(* LS Electric XG5000 project: OnlineHelp_ECAT_Example *)
(* This project contains various examples from the online help topics. *)
(* PLC LSPLC *)
(* module base 0 slot 0: Input/Output Module:XEM-DN/DP32HP (DC 24V Input, Transistor Output, 32 Contacts) *)
(* module base 0 slot 1: Internal Positioning:XBF-PO06E (Open Collector Type, 6 Axis) *)
(* module base 0 slot 2: Positioning Module:XBF-PN08B (Position Control, EtherCAT Network Type(8 axis)) *)
VAR_GLOBAL
    _0002_A1_RDY AT %UX0.2.0 : BOOL; (* Positioning Module: 1-Axis Ready *)
    _0002_A2_RDY AT %UX0.2.1 : BOOL; (* Positioning Module: 2-Axis Ready *)
    _0002_A3_RDY AT %UX0.2.2 : BOOL; (* Positioning Module: 3-Axis Ready *)
    _0002_A4_RDY AT %UX0.2.3 : BOOL; (* Positioning Module: 4-Axis Ready *)
    _0002_LINKUP_INFO AT %UX0.2.14 : BOOL; (* Positioning Module: Link up/down information *)
END_VAR

PROGRAM LP606_XPM_ECON_DCON_Example (* task: Scan Program *)
VAR
    Connect_Servos : BOOL; (* command to connect to ECAT servos *)
    DCON_FB : XPM_DCON; (* EtherCAT disconnect function block *)
    Disconnect_Servos : BOOL; (* Disconnect from ECAT servos *)
    ECON_FB : XPM_ECON; (* EtherCAT Connect function block. *)
END_VAR

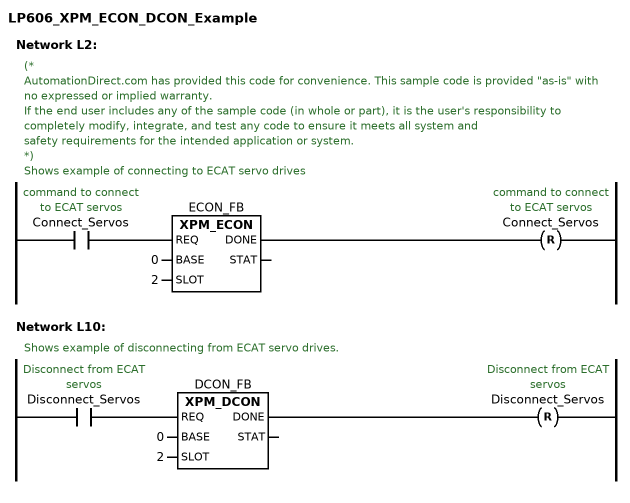
(* ( * / AutomationDirect.com has provided this code for convenience. This sample code is provided "as-is" with no expressed or implied warranty. / If the end user includes any of the sample code (in whole or part), it is the user's responsibility to completely modify, integrate, and test any code to ensure it meets all system and / safety requirements for the intended application or system. / * ) *)
(* Shows example of connecting to ECAT servo drives *)
(* Rung L2 *)
ECON_FB(REQ := Connect_Servos, BASE := 0, SLOT := 2);
IF ECON_FB.DONE THEN Connect_Servos := FALSE; END_IF;
(* Shows example of disconnecting from ECAT servo drives. *)
(* Rung L10 *)
DCON_FB(REQ := Disconnect_Servos, BASE := 0, SLOT := 2);
IF DCON_FB.DONE THEN Disconnect_Servos := FALSE; END_IF;
END_PROGRAM

PROGRAM LP607_XPM_SVON_SVOFF_Example (* task: Scan Program *)
(* This is an example for LP605 *)
VAR
    Axis1_SVOFF : XPM_SVOFF; (* function block for axis 1 servo off *)
    Axis1_SVOFF_Cmd : BOOL; (* axis 1 servo off command *)
    Axis1_SVON : XPM_SVON; (* SVON fb for axis 1 *)
    Axis1_SVON_Cmd : BOOL; (* axis 1 servo on command *)
END_VAR
VAR_EXTERNAL
    _0002_A1_RDY : BOOL; (* AT %UX0.2.0 *) (* Positioning Module: 1-Axis Ready *)
    _0002_LINKUP_INFO : BOOL; (* AT %UX0.2.14 *) (* Positioning Module: Link up/down information *)
END_VAR

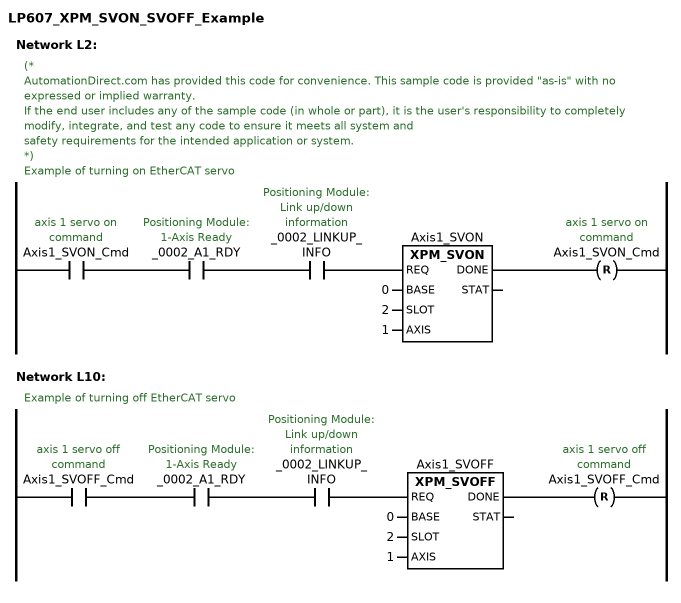
(* ( * / AutomationDirect.com has provided this code for convenience. This sample code is provided "as-is" with no expressed or implied warranty. / If the end user includes any of the sample code (in whole or part), it is the user's responsibility to completely modify, integrate, and test any code to ensure it meets all system and / safety requirements for the intended application or system. / * ) *)
(* Example of turning on EtherCAT servo *)
(* Rung L2 *)
Axis1_SVON(REQ := Axis1_SVON_Cmd AND _0002_A1_RDY AND _0002_LINKUP_INFO, BASE := 0, SLOT := 2, AXIS := 1);
IF Axis1_SVON.DONE THEN Axis1_SVON_Cmd := FALSE; END_IF;
(* Example of turning off EtherCAT servo *)
(* Rung L10 *)
Axis1_SVOFF(REQ := Axis1_SVOFF_Cmd AND _0002_A1_RDY AND _0002_LINKUP_INFO, BASE := 0, SLOT := 2, AXIS := 1);
IF Axis1_SVOFF.DONE THEN Axis1_SVOFF_Cmd := FALSE; END_IF;
END_PROGRAM

PROGRAM LP608_XPM_SVERD_SRST_Example (* task: Scan Program *)
(* this is an example of XPM_SVERD and XPM_SRST function blocks *)
VAR
    Axis1_Error : UINT; (* store axis 1 error *)
    Axis1_SRST : XPM_SRST; (* XPM_SRST for axis 1 *)
    Axis1_SVERD : XPM_SVERD; (* servo error reading for axis 1 *)
    Read_Axis1_Error : BOOL; (* command to read axis 1 error *)
    Reset_Axis1_Error : BOOL; (* reset command for axis error *)
END_VAR

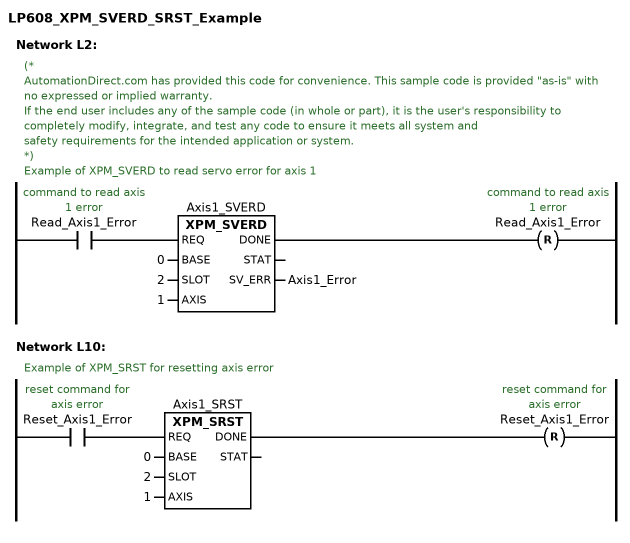
(* ( * / AutomationDirect.com has provided this code for convenience. This sample code is provided "as-is" with no expressed or implied warranty. / If the end user includes any of the sample code (in whole or part), it is the user's responsibility to completely modify, integrate, and test any code to ensure it meets all system and / safety requirements for the intended application or system. / * ) *)
(* Example of XPM_SVERD to read servo error for axis 1 *)
(* Rung L2 *)
Axis1_SVERD(REQ := Read_Axis1_Error, BASE := 0, SLOT := 2, AXIS := 1, SV_ERR => Axis1_Error);
IF Axis1_SVERD.DONE THEN Read_Axis1_Error := FALSE; END_IF;
(* Example of XPM_SRST for resetting axis error *)
(* Rung L10 *)
Axis1_SRST(REQ := Reset_Axis1_Error, BASE := 0, SLOT := 2, AXIS := 1);
IF Axis1_SRST.DONE THEN Reset_Axis1_Error := FALSE; END_IF;
END_PROGRAM

PROGRAM LP611_XPM_ENCRD_Example (* task: Scan Program *)
(* example for LP607 encoder reading *)
VAR
    Encoder_FB : XPM_ENCRD; (* reading encoder value *)
    Encoder_Value : DINT; (* encoder value from the read *)
    Read_Encoder_Value : BOOL; (* command to read encoder value. *)
END_VAR
VAR_EXTERNAL
    _0002_A1_RDY : BOOL; (* AT %UX0.2.0 *) (* Positioning Module: 1-Axis Ready *)
    _0002_LINKUP_INFO : BOOL; (* AT %UX0.2.14 *) (* Positioning Module: Link up/down information *)
END_VAR

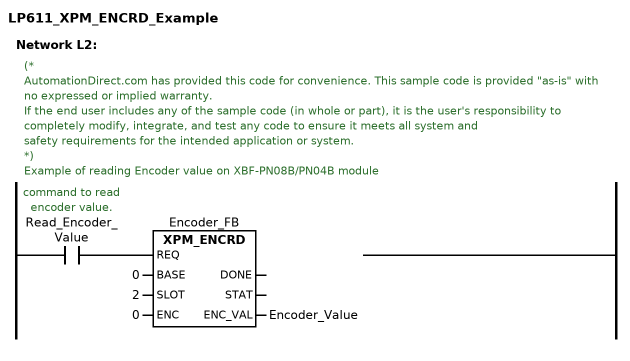
(* ( * / AutomationDirect.com has provided this code for convenience. This sample code is provided "as-is" with no expressed or implied warranty. / If the end user includes any of the sample code (in whole or part), it is the user's responsibility to completely modify, integrate, and test any code to ensure it meets all system and / safety requirements for the intended application or system. / * ) *)
(* Example of reading Encoder value on XBF-PN08B/PN04B module *)
(* Rung L2 *)
Encoder_FB(REQ := Read_Encoder_Value, BASE := 0, SLOT := 2, ENC := 0, ENC_VAL => Encoder_Value);
END_PROGRAM

PROGRAM LP612_XPM_TRQ_Example (* task: Scan Program *)
(* this is an example of XPM_TRQ *)
VAR
    Axes_SVOFF_Cmd : BOOL; (* axis 1 servo off command *)
    Axes_SVON_Cmd : BOOL; (* axes servo on command *)
    Axis1_Home : XPM_FLT; (* direct home of axis 1 *)
    Axis1_SVOFF : XPM_SVOFF; (* function block for axis 1 servo off *)
    Axis1_SVON : XPM_SVON; (* SVON fb for axis 1 *)
    Axis1_Torque_Time : UINT; (* gradient time for axis 1 torque fb *)
    Axis1_Torque_Value : INT; (* torque value for axis 1 *)
    Connect_Servos : BOOL; (* command to connect to ECAT servos *)
    DCON_FB : XPM_DCON; (* EtherCAT disconnect FB *)
    Disconnect_Servos : BOOL; (* Disconnect from ECAT servos *)
    ECON_FB : XPM_ECON; (* EtherCAT connect FB *)
    Execute_Torque_Control : BOOL; (* command to execute torque control *)
    Home_Axes : BOOL; (* home the axes *)
    TorqueCtrl_FB : XPM_TRQ; (* torque control fb for axis 1 *)
END_VAR
VAR_EXTERNAL
    _0002_A1_RDY : BOOL; (* AT %UX0.2.0 *) (* Positioning Module: 1-Axis Ready *)
    _0002_A4_RDY : BOOL; (* AT %UX0.2.3 *) (* Positioning Module: 4-Axis Ready *)
    _0002_LINKUP_INFO : BOOL; (* AT %UX0.2.14 *) (* Positioning Module: Link up/down information *)
END_VAR

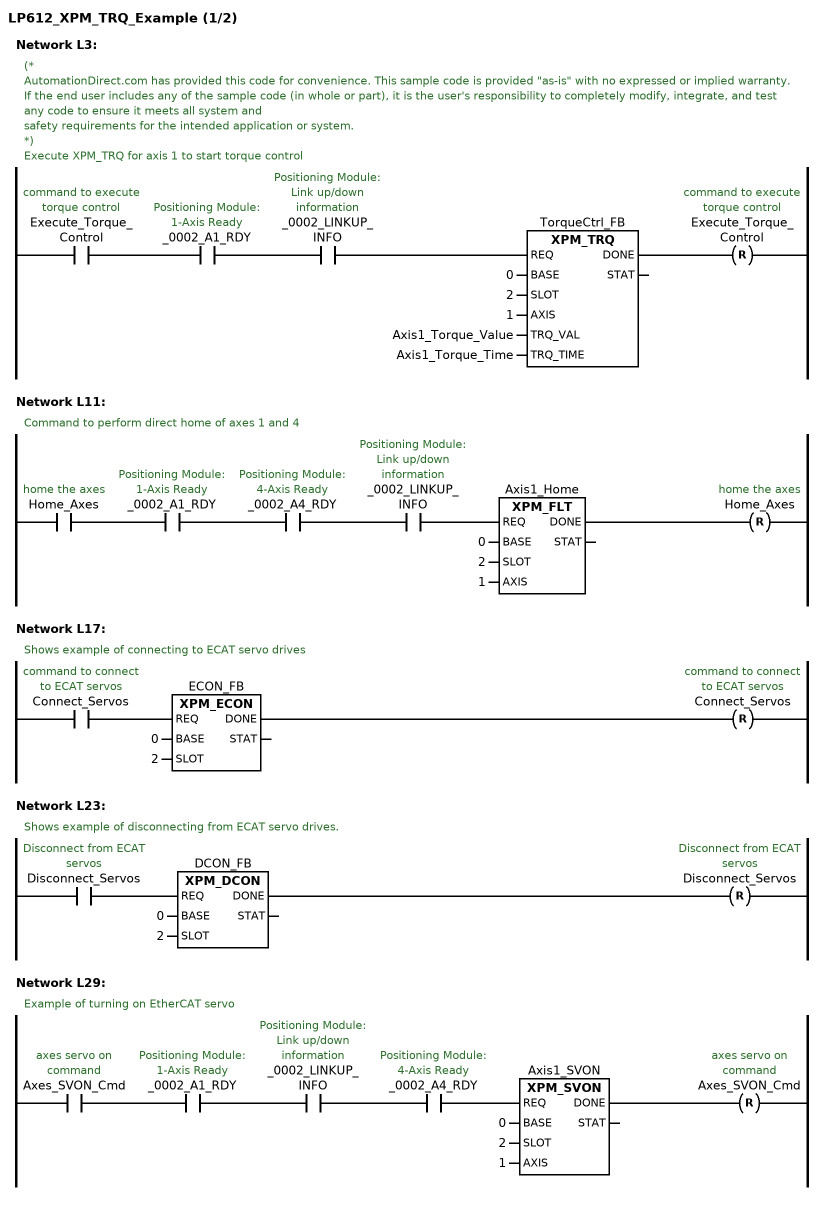
(* ( * / AutomationDirect.com has provided this code for convenience. This sample code is provided "as-is" with no expressed or implied warranty. / If the end user includes any of the sample code (in whole or part), it is the user's responsibility to completely modify, integrate, and test any code to ensure it meets all system and / safety requirements for the intended application or system. / * ) *)
(* Execute XPM_TRQ for axis 1 to start torque control *)
(* Rung L3 *)
TorqueCtrl_FB(REQ := Execute_Torque_Control AND _0002_A1_RDY AND _0002_LINKUP_INFO, BASE := 0, SLOT := 2, AXIS := 1, TRQ_VAL := Axis1_Torque_Value, TRQ_TIME := Axis1_Torque_Time);
IF TorqueCtrl_FB.DONE THEN Execute_Torque_Control := FALSE; END_IF;
(* Command to perform direct home of axes 1 and 4 *)
(* Rung L11 *)
Axis1_Home(REQ := Home_Axes AND _0002_A1_RDY AND _0002_A4_RDY AND _0002_LINKUP_INFO, BASE := 0, SLOT := 2, AXIS := 1);
IF Axis1_Home.DONE THEN Home_Axes := FALSE; END_IF;
(* Shows example of connecting to ECAT servo drives *)
(* Rung L17 *)
ECON_FB(REQ := Connect_Servos, BASE := 0, SLOT := 2);
IF ECON_FB.DONE THEN Connect_Servos := FALSE; END_IF;
(* Shows example of disconnecting from ECAT servo drives. *)
(* Rung L23 *)
DCON_FB(REQ := Disconnect_Servos, BASE := 0, SLOT := 2);
IF DCON_FB.DONE THEN Disconnect_Servos := FALSE; END_IF;
(* Example of turning on EtherCAT servo *)
(* Rung L29 *)
Axis1_SVON(REQ := Axes_SVON_Cmd AND _0002_A1_RDY AND _0002_LINKUP_INFO AND _0002_A4_RDY, BASE := 0, SLOT := 2, AXIS := 1);
IF Axis1_SVON.DONE THEN Axes_SVON_Cmd := FALSE; END_IF;

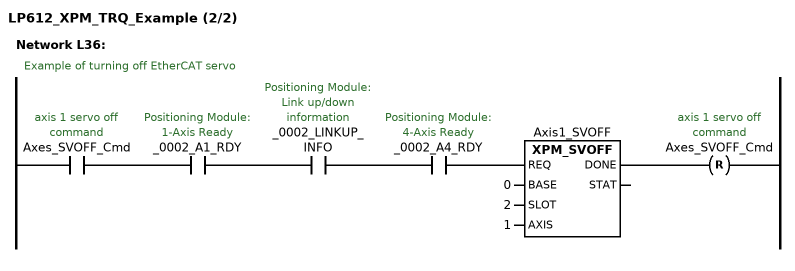
(* Example of turning off EtherCAT servo *)
(* Rung L36 *)
Axis1_SVOFF(REQ := Axes_SVOFF_Cmd AND _0002_A1_RDY AND _0002_LINKUP_INFO AND _0002_A4_RDY, BASE := 0, SLOT := 2, AXIS := 1);
IF Axis1_SVOFF.DONE THEN Axes_SVOFF_Cmd := FALSE; END_IF;
END_PROGRAM

PROGRAM LP613_XPM_SVPRD_SVPWR_SVSAVE_Example (* task: Scan Program *)
(* this is an example program for fbs XPM_SVPRD, XPM_SVPWR, XPM_SVSAVE *)
VAR
    Axis1_SVPRD : XPM_SVPRD; (* fb for read parameter read for axis 1 *)
    Axis1_SVPRD2 : XPM_SVPRD; (* reading Home offset after writing to it *)
    Axis1_SVPWR : XPM_SVPWR; (* XPM_SVPWR fb *)
    Axis1_SVSAVE : XPM_SVSAVE; (* axis 1 fb to save parameters *)
    Execute_Parameter_Read : BOOL; (* command to execute servo parameter read *)
    Execute_Parameter_Read2 : BOOL; (* used to read home offset after writing to it *)
    Execute_Parameter_Save : BOOL; (* command to execute parameter save on servo *)
    Execute_Parameter_Write : BOOL; (* command to write parameter data *)
    ParameterRead_Data : DINT; (* store parameter read data *)
    ParameterWrite_Data : DINT; (* data to write to a parameter *)
    SAVE_AXIS : USINT; (* save axis parameter of XPM_SVSAVE fb *)
END_VAR
VAR_EXTERNAL
    _0002_A1_RDY : BOOL; (* AT %UX0.2.0 *) (* Positioning Module: 1-Axis Ready *)
    _0002_LINKUP_INFO : BOOL; (* AT %UX0.2.14 *) (* Positioning Module: Link up/down information *)
END_VAR

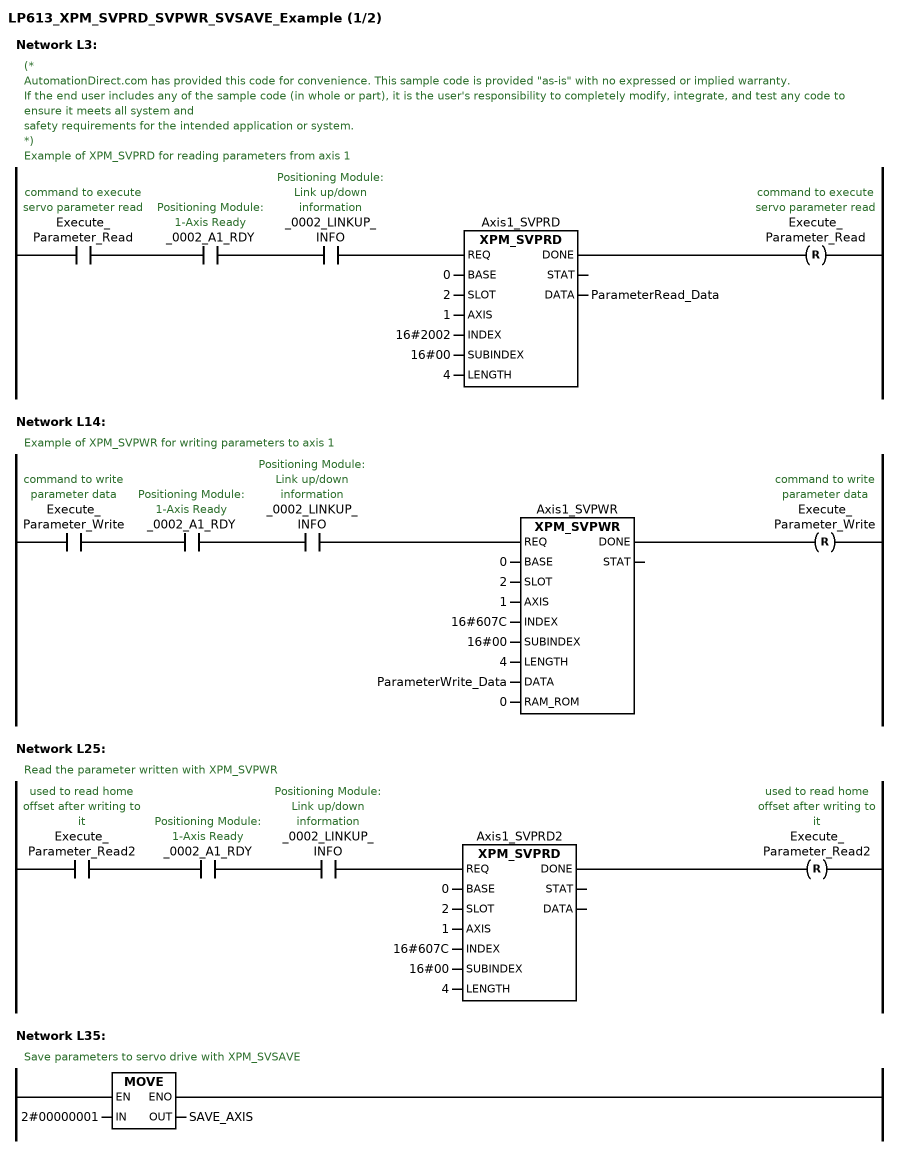
(* ( * / AutomationDirect.com has provided this code for convenience. This sample code is provided "as-is" with no expressed or implied warranty. / If the end user includes any of the sample code (in whole or part), it is the user's responsibility to completely modify, integrate, and test any code to ensure it meets all system and / safety requirements for the intended application or system. / * ) *)
(* Example of XPM_SVPRD for reading parameters from axis 1 *)
(* Rung L3 *)
Axis1_SVPRD(REQ := Execute_Parameter_Read AND _0002_A1_RDY AND _0002_LINKUP_INFO, BASE := 0, SLOT := 2, AXIS := 1, INDEX := 16#2002, SUBINDEX := 16#00, LENGTH := 4, DATA => ParameterRead_Data);
IF Axis1_SVPRD.DONE THEN Execute_Parameter_Read := FALSE; END_IF;
(* Example of XPM_SVPWR for writing parameters to axis 1 *)
(* Rung L14 *)
Axis1_SVPWR(REQ := Execute_Parameter_Write AND _0002_A1_RDY AND _0002_LINKUP_INFO, BASE := 0, SLOT := 2, AXIS := 1, INDEX := 16#607C, SUBINDEX := 16#00, LENGTH := 4, DATA := ParameterWrite_Data, RAM_ROM := 0);
IF Axis1_SVPWR.DONE THEN Execute_Parameter_Write := FALSE; END_IF;
(* Read the parameter written with XPM_SVPWR *)
(* Rung L25 *)
Axis1_SVPRD2(REQ := Execute_Parameter_Read2 AND _0002_A1_RDY AND _0002_LINKUP_INFO, BASE := 0, SLOT := 2, AXIS := 1, INDEX := 16#607C, SUBINDEX := 16#00, LENGTH := 4);
IF Axis1_SVPRD2.DONE THEN Execute_Parameter_Read2 := FALSE; END_IF;
(* Save parameters to servo drive with XPM_SVSAVE *)
(* Rung L35 *)
SAVE_AXIS := 2#00000001;

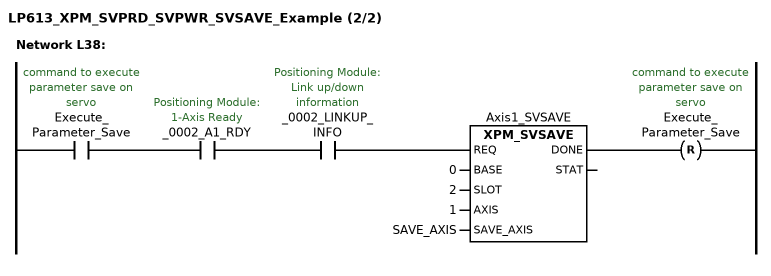
(* Rung L38 *)
Axis1_SVSAVE(REQ := Execute_Parameter_Save AND _0002_A1_RDY AND _0002_LINKUP_INFO, BASE := 0, SLOT := 2, AXIS := 1, SAVE_AXIS := SAVE_AXIS);
IF Axis1_SVSAVE.DONE THEN Execute_Parameter_Save := FALSE; END_IF;
END_PROGRAM

PROGRAM LP614_Position_Latch_Examples (* task: Scan Program *)
(* example program for XPM_LSET, XPM_LRD, XPM_LCLR  function blocks *)
VAR
    Axes_SVOFF_Cmd : BOOL; (* axis 1 servo off command *)
    Axes_SVON_Cmd : BOOL; (* axes servo on command *)
    Axis1_DST : XPM_DST; (* direct start for axis 4 *)
    Axis1_Home : XPM_FLT; (* direct home of axis 1 *)
    Axis1_LCLR_Cmd : BOOL; (* run latch clear position *)
    Axis1_LCNT : UINT; (* axis 1 l_cnt variable *)
    Axis1_LData : ARRAY[0..9] OF DINT; (* LDATA for axis 1 XPM_LRD fb *)
    Axis1_LRD_Cmd : BOOL; (* command to read latch position on axis 1 *)
    Axis1_LSET_Cmd : BOOL; (* command to run XPM_LSET *)
    Axis1_Speed_Cmd : BOOL; (* command to perform speed move *)
    Axis1_SVOFF : XPM_SVOFF; (* function block for axis 1 servo off *)
    Axis1_SVON : XPM_SVON; (* SVON fb for axis 1 *)
    Axis1_XPM_LCLR : XPM_LCLR; (* axis 1 XPM_LCLR fb *)
    Axis1_XPM_LRD : XPM_LRD; (* axis 1 xpm_lrd fb *)
    Axis1_XPM_LSET : XPM_LSET; (* xpm lset fb *)
    Connect_Servos : BOOL; (* command to connect to ECAT servos *)
    DCON_FB : XPM_DCON; (* EtherCAT disconnect fb *)
    Disconnect_Servos : BOOL; (* Disconnect from ECAT servos *)
    ECON_FB : XPM_ECON; (* EtherCAT connect fb *)
    Home_Axes : BOOL; (* home the axes *)
END_VAR
VAR_EXTERNAL
    _0002_A1_RDY : BOOL; (* AT %UX0.2.0 *) (* Positioning Module: 1-Axis Ready *)
    _0002_LINKUP_INFO : BOOL; (* AT %UX0.2.14 *) (* Positioning Module: Link up/down information *)
END_VAR

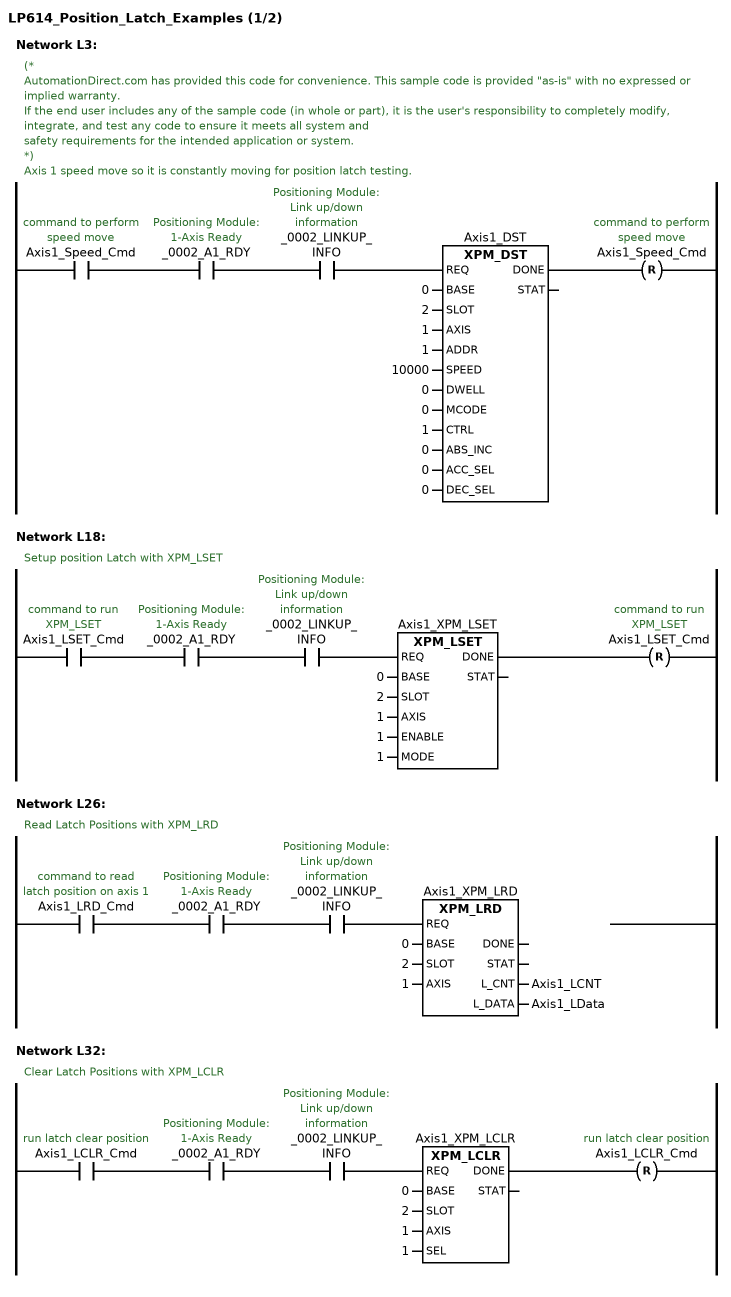
(* ( * / AutomationDirect.com has provided this code for convenience. This sample code is provided "as-is" with no expressed or implied warranty. / If the end user includes any of the sample code (in whole or part), it is the user's responsibility to completely modify, integrate, and test any code to ensure it meets all system and / safety requirements for the intended application or system. / * ) *)
(* Axis 1 speed move so it is constantly moving for position latch testing. *)
(* Rung L3 *)
Axis1_DST(REQ := Axis1_Speed_Cmd AND _0002_A1_RDY AND _0002_LINKUP_INFO, BASE := 0, SLOT := 2, AXIS := 1, ADDR := 1, SPEED := 10000, DWELL := 0, MCODE := 0, CTRL := 1, ABS_INC := 0, ACC_SEL := 0, DEC_SEL := 0);
IF Axis1_DST.DONE THEN Axis1_Speed_Cmd := FALSE; END_IF;
(* Setup position Latch with XPM_LSET *)
(* Rung L18 *)
Axis1_XPM_LSET(REQ := Axis1_LSET_Cmd AND _0002_A1_RDY AND _0002_LINKUP_INFO, BASE := 0, SLOT := 2, AXIS := 1, ENABLE := 1, MODE := 1);
IF Axis1_XPM_LSET.DONE THEN Axis1_LSET_Cmd := FALSE; END_IF;
(* Read Latch Positions with XPM_LRD *)
(* Rung L26 *)
Axis1_XPM_LRD(REQ := Axis1_LRD_Cmd AND _0002_A1_RDY AND _0002_LINKUP_INFO, BASE := 0, SLOT := 2, AXIS := 1, L_CNT => Axis1_LCNT, L_DATA => Axis1_LData);
(* Clear Latch Positions with XPM_LCLR *)
(* Rung L32 *)
Axis1_XPM_LCLR(REQ := Axis1_LCLR_Cmd AND _0002_A1_RDY AND _0002_LINKUP_INFO, BASE := 0, SLOT := 2, AXIS := 1, SEL := 1);
IF Axis1_XPM_LCLR.DONE THEN Axis1_LCLR_Cmd := FALSE; END_IF;

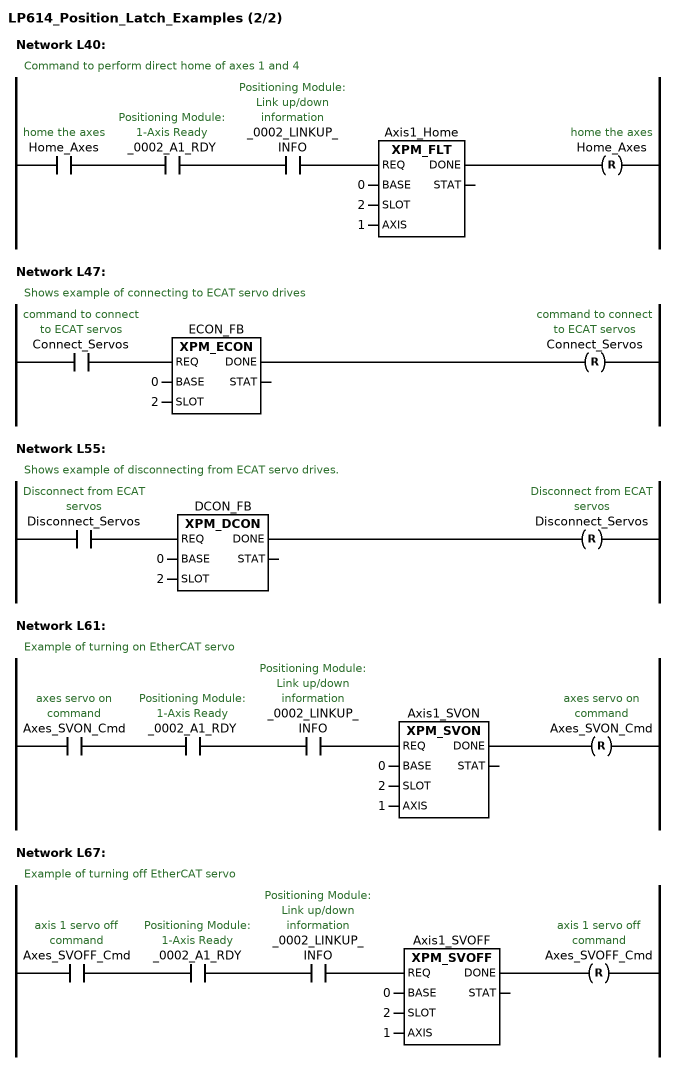
(* Command to perform direct home of axes 1 and 4 *)
(* Rung L40 *)
Axis1_Home(REQ := Home_Axes AND _0002_A1_RDY AND _0002_LINKUP_INFO, BASE := 0, SLOT := 2, AXIS := 1);
IF Axis1_Home.DONE THEN Home_Axes := FALSE; END_IF;
(* Shows example of connecting to ECAT servo drives *)
(* Rung L47 *)
ECON_FB(REQ := Connect_Servos, BASE := 0, SLOT := 2);
IF ECON_FB.DONE THEN Connect_Servos := FALSE; END_IF;
(* Shows example of disconnecting from ECAT servo drives. *)
(* Rung L55 *)
DCON_FB(REQ := Disconnect_Servos, BASE := 0, SLOT := 2);
IF DCON_FB.DONE THEN Disconnect_Servos := FALSE; END_IF;
(* Example of turning on EtherCAT servo *)
(* Rung L61 *)
Axis1_SVON(REQ := Axes_SVON_Cmd AND _0002_A1_RDY AND _0002_LINKUP_INFO, BASE := 0, SLOT := 2, AXIS := 1);
IF Axis1_SVON.DONE THEN Axes_SVON_Cmd := FALSE; END_IF;
(* Example of turning off EtherCAT servo *)
(* Rung L67 *)
Axis1_SVOFF(REQ := Axes_SVOFF_Cmd AND _0002_A1_RDY AND _0002_LINKUP_INFO, BASE := 0, SLOT := 2, AXIS := 1);
IF Axis1_SVOFF.DONE THEN Axes_SVOFF_Cmd := FALSE; END_IF;
END_PROGRAM

PROGRAM LP615_XPM_SSSD_SSSPD_Example (* task: Scan Program *)
(* example program for XPM_SSSD and XPM_SSSPD function blocks. *)
VAR
    Axes_SVOFF_Cmd : BOOL; (* axis 1 servo off command *)
    Axes_SVON_Cmd : BOOL; (* axes servo on command *)
    Axis1_Home : XPM_FLT; (* direct home of axis 1 *)
    Axis1_SSSD : XPM_SSSD; (* XPM_SSSD fb for axis 1 *)
    Axis1_SSSPD : XPM_SSSPD; (* XPM_SSSPD fb for axis 1 *)
    Axis1_SVOFF : XPM_SVOFF; (* function block for axis 1 servo off *)
    Axis1_SVON : XPM_SVON; (* SVON fb for axis 1 *)
    Axis1_Sync_CMD1 : BOOL; (* command to perform XPM_SSSD fb *)
    Axis1_Sync_CMD2 : BOOL; (* command for XPM_SSSPD fb *)
    Axis4_DST : XPM_DST; (* direct start for axis 4 *)
    Axis4_Home : XPM_FLT; (* direct home axis 4 *)
    Axis4_SVOFF : XPM_SVOFF; (* servo off fb for axis 4 *)
    Axis4_SVON : XPM_SVON; (* servo on fb for axis 4 *)
    Connect_Servos : BOOL; (* command to connect to ECAT servos *)
    DCON_FB : XPM_DCON; (* EtherCAT disconnect FB *)
    Disconnect_Servos : BOOL; (* Disconnect from ECAT servos *)
    ECON_FB : XPM_ECON; (* EtherCAT connect fb *)
    Home_Axes : BOOL; (* home the axes *)
END_VAR
VAR_EXTERNAL
    _0002_A1_RDY : BOOL; (* AT %UX0.2.0 *) (* Positioning Module: 1-Axis Ready *)
    _0002_A4_RDY : BOOL; (* AT %UX0.2.3 *) (* Positioning Module: 4-Axis Ready *)
    _0002_LINKUP_INFO : BOOL; (* AT %UX0.2.14 *) (* Positioning Module: Link up/down information *)
END_VAR
VAR
    _p1 : BOOL;
    _p2 : BOOL;
    _p3 : BOOL;
END_VAR

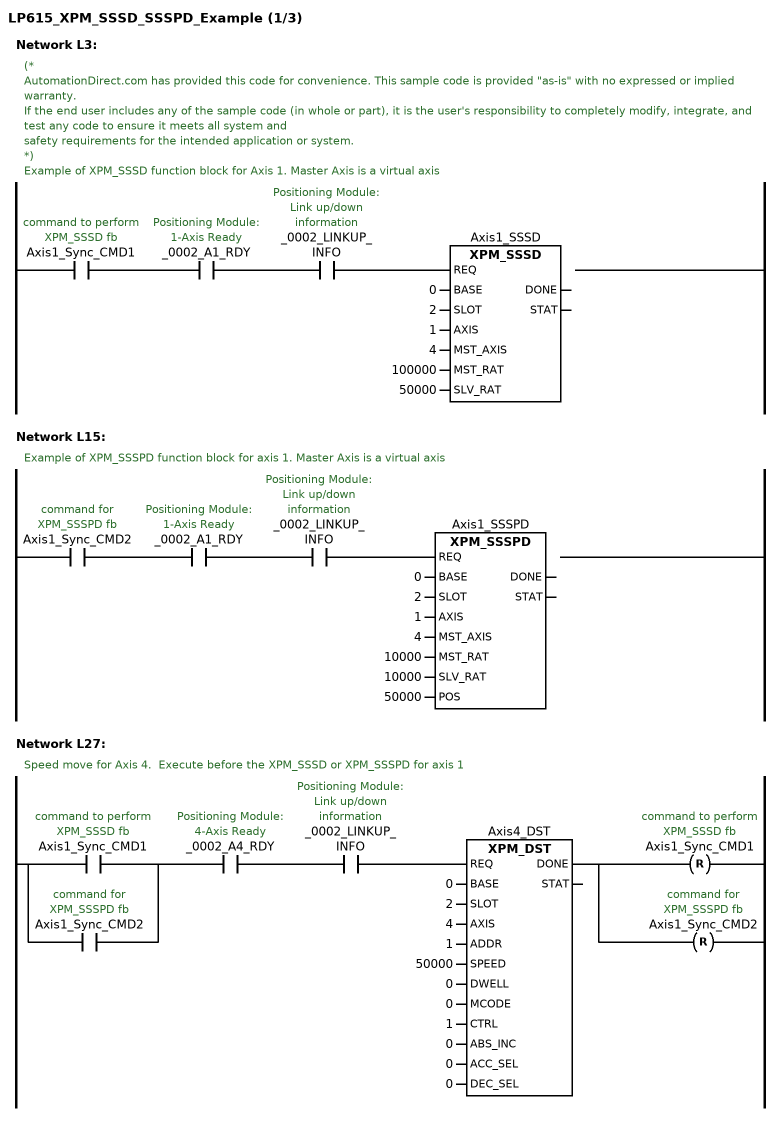
(* ( * / AutomationDirect.com has provided this code for convenience. This sample code is provided "as-is" with no expressed or implied warranty. / If the end user includes any of the sample code (in whole or part), it is the user's responsibility to completely modify, integrate, and test any code to ensure it meets all system and / safety requirements for the intended application or system. / * ) *)
(* Example of XPM_SSSD function block for Axis 1. Master Axis is a virtual axis *)
(* Rung L3 *)
Axis1_SSSD(REQ := Axis1_Sync_CMD1 AND _0002_A1_RDY AND _0002_LINKUP_INFO, BASE := 0, SLOT := 2, AXIS := 1, MST_AXIS := 4, MST_RAT := 100000, SLV_RAT := 50000);
(* Example of XPM_SSSPD function block for axis 1. Master Axis is a virtual axis *)
(* Rung L15 *)
Axis1_SSSPD(REQ := Axis1_Sync_CMD2 AND _0002_A1_RDY AND _0002_LINKUP_INFO, BASE := 0, SLOT := 2, AXIS := 1, MST_AXIS := 4, MST_RAT := 10000, SLV_RAT := 10000, POS := 50000);
(* Speed move for Axis 4.  Execute before the XPM_SSSD or XPM_SSSPD for axis 1 *)
(* Rung L27 *)
Axis4_DST(REQ := (Axis1_Sync_CMD1 OR Axis1_Sync_CMD2) AND _0002_A4_RDY AND _0002_LINKUP_INFO, BASE := 0, SLOT := 2, AXIS := 4, ADDR := 1, SPEED := 50000, DWELL := 0, MCODE := 0, CTRL := 1, ABS_INC := 0, ACC_SEL := 0, DEC_SEL := 0);
IF Axis4_DST.DONE THEN
    Axis1_Sync_CMD1 := FALSE;
    Axis1_Sync_CMD2 := FALSE;
END_IF;

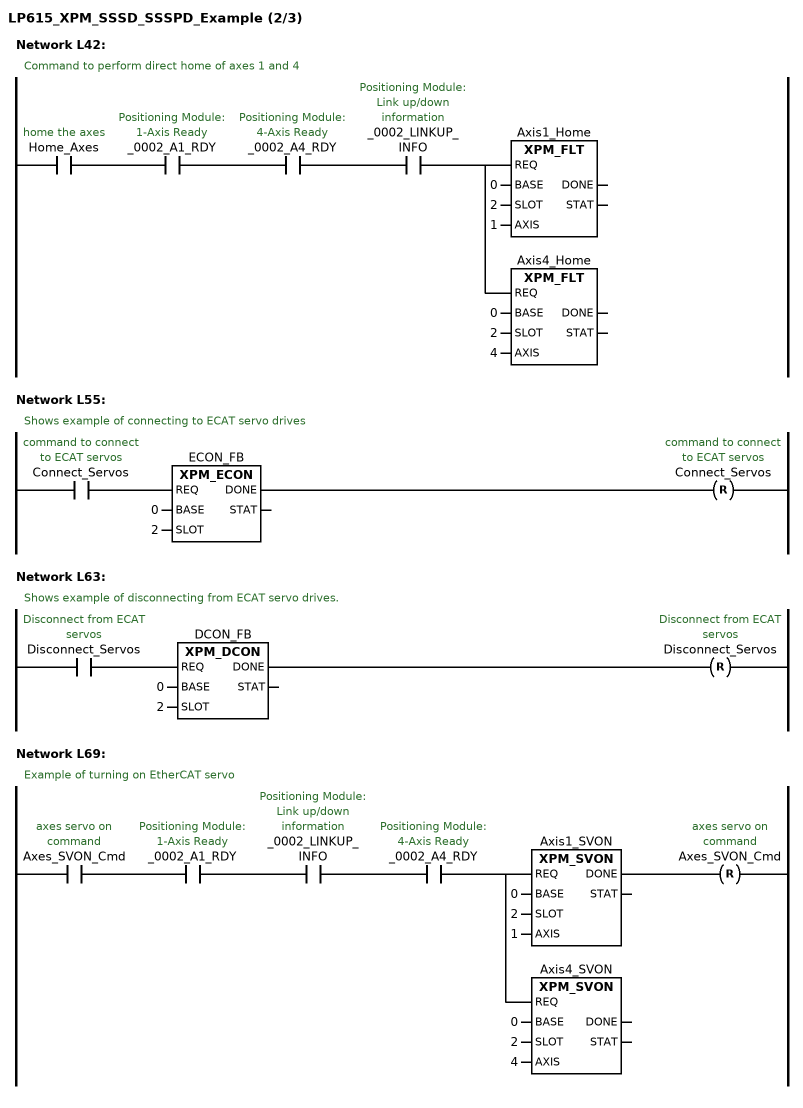
(* Command to perform direct home of axes 1 and 4 *)
(* Rung L42 *)
_p1 := Home_Axes AND _0002_A1_RDY AND _0002_A4_RDY AND _0002_LINKUP_INFO;
Axis1_Home(REQ := _p1, BASE := 0, SLOT := 2, AXIS := 1);
Axis4_Home(REQ := _p1, BASE := 0, SLOT := 2, AXIS := 4);
(* Shows example of connecting to ECAT servo drives *)
(* Rung L55 *)
ECON_FB(REQ := Connect_Servos, BASE := 0, SLOT := 2);
IF ECON_FB.DONE THEN Connect_Servos := FALSE; END_IF;
(* Shows example of disconnecting from ECAT servo drives. *)
(* Rung L63 *)
DCON_FB(REQ := Disconnect_Servos, BASE := 0, SLOT := 2);
IF DCON_FB.DONE THEN Disconnect_Servos := FALSE; END_IF;
(* Example of turning on EtherCAT servo *)
(* Rung L69 *)
_p2 := Axes_SVON_Cmd AND _0002_A1_RDY AND _0002_LINKUP_INFO AND _0002_A4_RDY;
Axis1_SVON(REQ := _p2, BASE := 0, SLOT := 2, AXIS := 1);
IF Axis1_SVON.DONE THEN Axes_SVON_Cmd := FALSE; END_IF;
Axis4_SVON(REQ := _p2, BASE := 0, SLOT := 2, AXIS := 4);

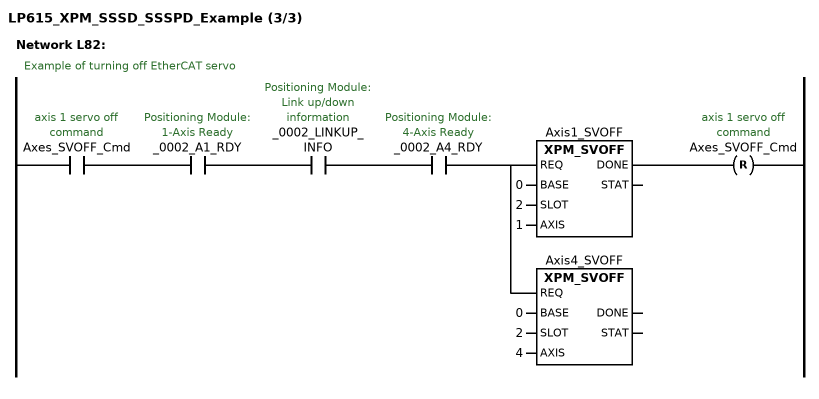
(* Example of turning off EtherCAT servo *)
(* Rung L82 *)
_p3 := Axes_SVOFF_Cmd AND _0002_A1_RDY AND _0002_LINKUP_INFO AND _0002_A4_RDY;
Axis1_SVOFF(REQ := _p3, BASE := 0, SLOT := 2, AXIS := 1);
IF Axis1_SVOFF.DONE THEN Axes_SVOFF_Cmd := FALSE; END_IF;
Axis4_SVOFF(REQ := _p3, BASE := 0, SLOT := 2, AXIS := 4);
END_PROGRAM

PROGRAM LP616_XPM_PHASING_Example (* task: Scan Program *)
(* example program for XPM_PHASING  function block. *)
VAR
    Axes_SVOFF_Cmd : BOOL; (* axis 1 servo off command *)
    Axes_SVON_Cmd : BOOL; (* axes servo on command *)
    Axis1_Home : XPM_FLT; (* direct home of axis 1 *)
    Axis1_Phase_CMD : BOOL; (* command to perform XPM_PHASING fb *)
    Axis1_Phase_Value : DINT; (* phase correction value *)
    Axis1_Phase_Velocity : UDINT; (* velocity of axis 1 phasing move *)
    Axis1_Phasing : XPM_PHASING; (* XPM_PHASING fb for axis 1 *)
    Axis1_SSSPD : XPM_SSSPD; (* XPM_SSSPD fb for axis 1 *)
    Axis1_SVOFF : XPM_SVOFF; (* function block for axis 1 servo off *)
    Axis1_SVON : XPM_SVON; (* SVON fb for axis 1 *)
    Axis1_Sync_CMD : BOOL; (* command for XPM_SSSPD fb *)
    Axis1_XPM_SSSD : XPM_SSSD; (* Axis 1 XPM_SSSD fb *)
    Axis4_DST : XPM_DST; (* direct start for axis 4 *)
    Axis4_Home : XPM_FLT; (* direct home axis 4 *)
    Axis4_SVOFF : XPM_SVOFF; (* servo off fb for axis 4 *)
    Axis4_SVON : XPM_SVON; (* servo on fb for axis 4 *)
    Connect_Servos : BOOL; (* command to connect to ECAT servos *)
    DCON_FB : XPM_DCON; (* EtherCAT disconnect FB *)
    Disconnect_Servos : BOOL; (* Disconnect from ECAT servos *)
    ECON_FB : XPM_ECON; (* EtherCAT connect FB *)
    Home_Axes : BOOL; (* home the axes *)
END_VAR
VAR_EXTERNAL
    _0002_A1_RDY : BOOL; (* AT %UX0.2.0 *) (* Positioning Module: 1-Axis Ready *)
    _0002_A4_RDY : BOOL; (* AT %UX0.2.3 *) (* Positioning Module: 4-Axis Ready *)
    _0002_LINKUP_INFO : BOOL; (* AT %UX0.2.14 *) (* Positioning Module: Link up/down information *)
END_VAR
VAR
    _p1 : BOOL;
    _p2 : BOOL;
    _p3 : BOOL;
END_VAR

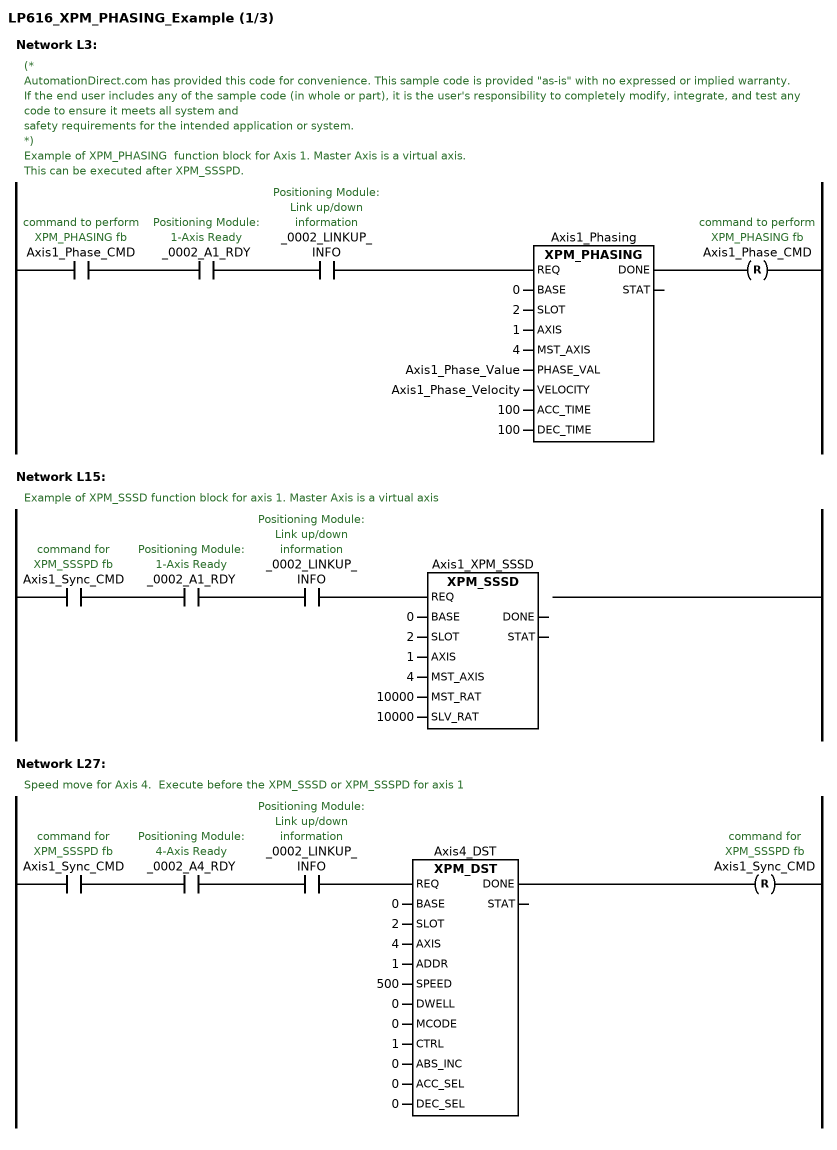
(* ( * / AutomationDirect.com has provided this code for convenience. This sample code is provided "as-is" with no expressed or implied warranty. / If the end user includes any of the sample code (in whole or part), it is the user's responsibility to completely modify, integrate, and test any code to ensure it meets all system and / safety requirements for the intended application or system. / * ) *)
(* Example of XPM_PHASING  function block for Axis 1. Master Axis is a virtual axis. / This can be executed after XPM_SSSPD. *)
(* Rung L3 *)
Axis1_Phasing(REQ := Axis1_Phase_CMD AND _0002_A1_RDY AND _0002_LINKUP_INFO, BASE := 0, SLOT := 2, AXIS := 1, MST_AXIS := 4, PHASE_VAL := Axis1_Phase_Value, VELOCITY := Axis1_Phase_Velocity, ACC_TIME := 100, DEC_TIME := 100);
IF Axis1_Phasing.DONE THEN Axis1_Phase_CMD := FALSE; END_IF;
(* Example of XPM_SSSD function block for axis 1. Master Axis is a virtual axis *)
(* Rung L15 *)
Axis1_XPM_SSSD(REQ := Axis1_Sync_CMD AND _0002_A1_RDY AND _0002_LINKUP_INFO, BASE := 0, SLOT := 2, AXIS := 1, MST_AXIS := 4, MST_RAT := 10000, SLV_RAT := 10000);
(* Speed move for Axis 4.  Execute before the XPM_SSSD or XPM_SSSPD for axis 1 *)
(* Rung L27 *)
Axis4_DST(REQ := Axis1_Sync_CMD AND _0002_A4_RDY AND _0002_LINKUP_INFO, BASE := 0, SLOT := 2, AXIS := 4, ADDR := 1, SPEED := 500, DWELL := 0, MCODE := 0, CTRL := 1, ABS_INC := 0, ACC_SEL := 0, DEC_SEL := 0);
IF Axis4_DST.DONE THEN Axis1_Sync_CMD := FALSE; END_IF;

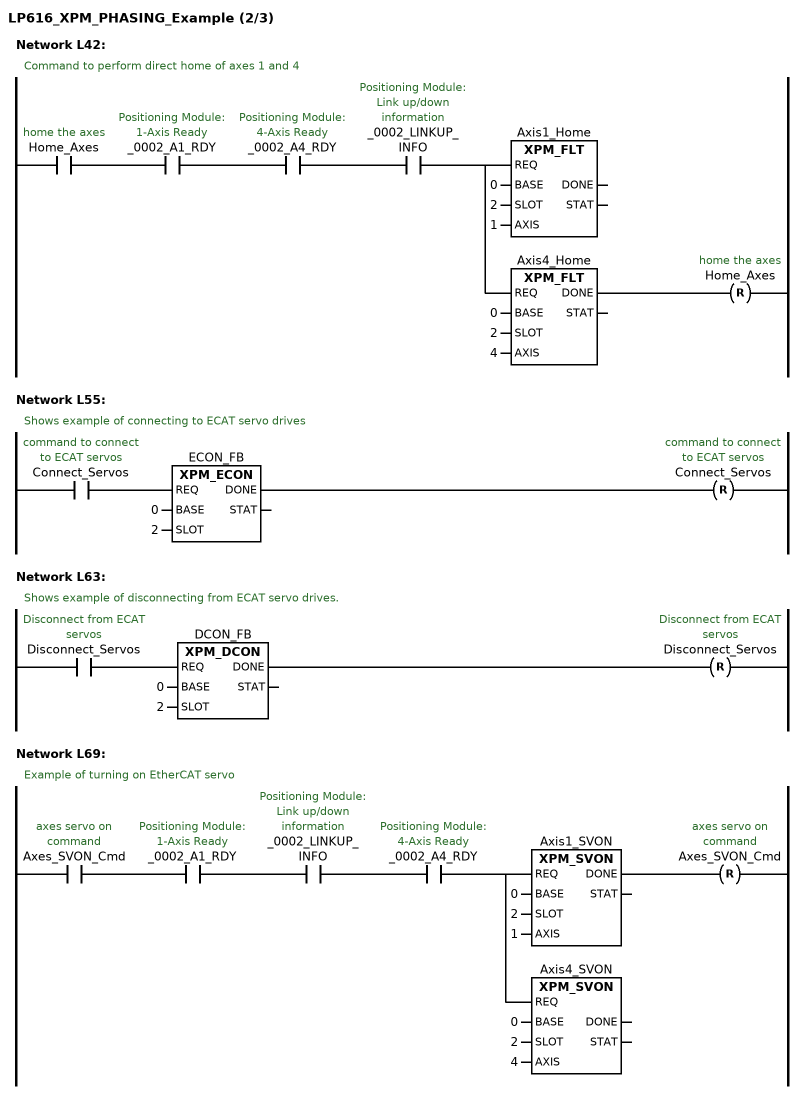
(* Command to perform direct home of axes 1 and 4 *)
(* Rung L42 *)
_p1 := Home_Axes AND _0002_A1_RDY AND _0002_A4_RDY AND _0002_LINKUP_INFO;
Axis1_Home(REQ := _p1, BASE := 0, SLOT := 2, AXIS := 1);
Axis4_Home(REQ := _p1, BASE := 0, SLOT := 2, AXIS := 4);
IF Axis4_Home.DONE THEN Home_Axes := FALSE; END_IF;
(* Shows example of connecting to ECAT servo drives *)
(* Rung L55 *)
ECON_FB(REQ := Connect_Servos, BASE := 0, SLOT := 2);
IF ECON_FB.DONE THEN Connect_Servos := FALSE; END_IF;
(* Shows example of disconnecting from ECAT servo drives. *)
(* Rung L63 *)
DCON_FB(REQ := Disconnect_Servos, BASE := 0, SLOT := 2);
IF DCON_FB.DONE THEN Disconnect_Servos := FALSE; END_IF;
(* Example of turning on EtherCAT servo *)
(* Rung L69 *)
_p2 := Axes_SVON_Cmd AND _0002_A1_RDY AND _0002_LINKUP_INFO AND _0002_A4_RDY;
Axis1_SVON(REQ := _p2, BASE := 0, SLOT := 2, AXIS := 1);
IF Axis1_SVON.DONE THEN Axes_SVON_Cmd := FALSE; END_IF;
Axis4_SVON(REQ := _p2, BASE := 0, SLOT := 2, AXIS := 4);

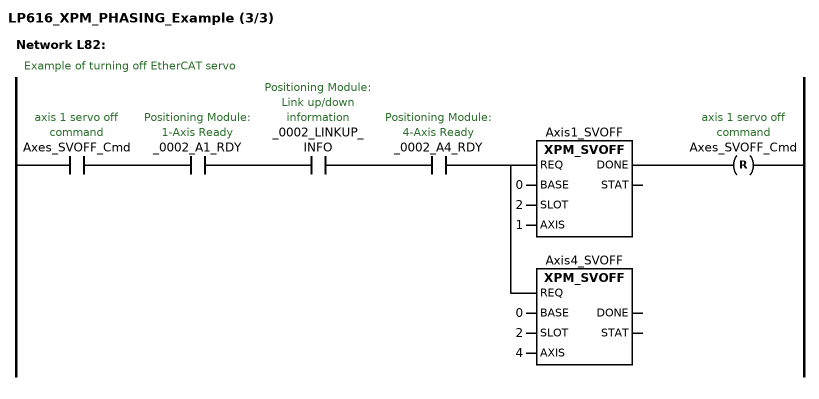
(* Example of turning off EtherCAT servo *)
(* Rung L82 *)
_p3 := Axes_SVOFF_Cmd AND _0002_A1_RDY AND _0002_LINKUP_INFO AND _0002_A4_RDY;
Axis1_SVOFF(REQ := _p3, BASE := 0, SLOT := 2, AXIS := 1);
IF Axis1_SVOFF.DONE THEN Axes_SVOFF_Cmd := FALSE; END_IF;
Axis4_SVOFF(REQ := _p3, BASE := 0, SLOT := 2, AXIS := 4);
END_PROGRAM

PROGRAM LP617_XPM_CAMA_Example (* task: Scan Program *)
(* example program for XPM_CAMA  function block. *)
VAR
    Axes_SVOFF_Cmd : BOOL; (* axis 1 servo off command *)
    Axes_SVON_Cmd : BOOL; (* axes servo on command *)
    Axis1_Home : XPM_FLT; (* direct home of axis 1 *)
    Axis1_SVOFF : XPM_SVOFF; (* function block for axis 1 servo off *)
    Axis1_SVON : XPM_SVON; (* SVON fb for axis 1 *)
    Axis1_XPM_CAMA : XPM_CAMA; (* XPM_CAMA fb for axis 1 *)
    Axis4_DST : XPM_DST; (* direct start for axis 4 *)
    Axis4_Home : XPM_FLT; (* direct home axis 4 *)
    Axis4_SVOFF : XPM_SVOFF; (* servo off fb for axis 4 *)
    Axis4_SVON : XPM_SVON; (* servo on fb for axis 4 *)
    Connect_Servos : BOOL; (* command to connect to ECAT servos *)
    DCON_FB : XPM_DCON; (* EtherCAT disconnect FB *)
    Disconnect_Servos : BOOL; (* Disconnect from ECAT servos *)
    ECON_FB : XPM_ECON; (* EtherCAT connect FB *)
    Home_Axes : BOOL; (* home the axes *)
    Run_Example : BOOL; (* command for running XPM_CAMA example. *)
END_VAR
VAR_EXTERNAL
    _0002_A1_RDY : BOOL; (* AT %UX0.2.0 *) (* Positioning Module: 1-Axis Ready *)
    _0002_A4_RDY : BOOL; (* AT %UX0.2.3 *) (* Positioning Module: 4-Axis Ready *)
    _0002_LINKUP_INFO : BOOL; (* AT %UX0.2.14 *) (* Positioning Module: Link up/down information *)
END_VAR
VAR
    _p1 : BOOL;
    _p2 : BOOL;
    _p3 : BOOL;
END_VAR

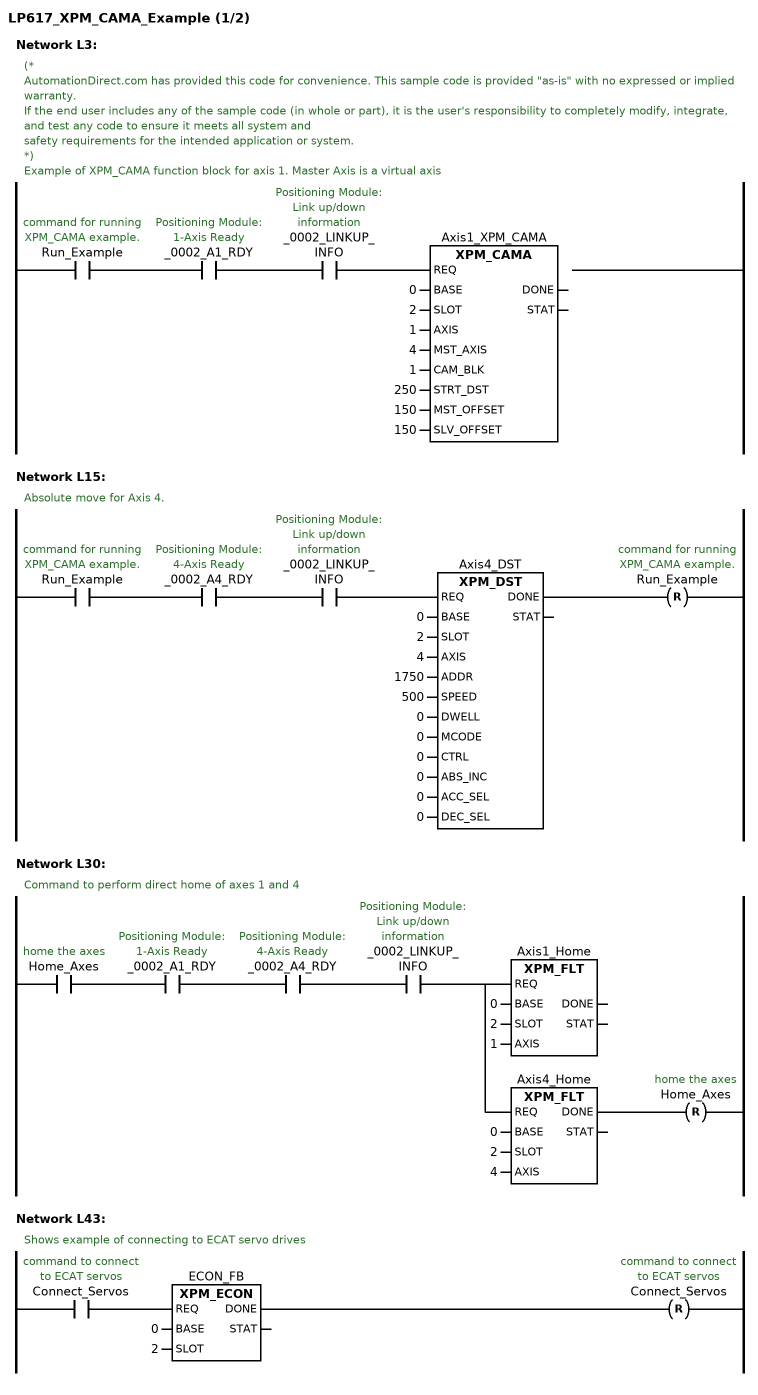
(* ( * / AutomationDirect.com has provided this code for convenience. This sample code is provided "as-is" with no expressed or implied warranty. / If the end user includes any of the sample code (in whole or part), it is the user's responsibility to completely modify, integrate, and test any code to ensure it meets all system and / safety requirements for the intended application or system. / * ) *)
(* Example of XPM_CAMA function block for axis 1. Master Axis is a virtual axis *)
(* Rung L3 *)
Axis1_XPM_CAMA(REQ := Run_Example AND _0002_A1_RDY AND _0002_LINKUP_INFO, BASE := 0, SLOT := 2, AXIS := 1, MST_AXIS := 4, CAM_BLK := 1, STRT_DST := 250, MST_OFFSET := 150, SLV_OFFSET := 150);
(* Absolute move for Axis 4. *)
(* Rung L15 *)
Axis4_DST(REQ := Run_Example AND _0002_A4_RDY AND _0002_LINKUP_INFO, BASE := 0, SLOT := 2, AXIS := 4, ADDR := 1750, SPEED := 500, DWELL := 0, MCODE := 0, CTRL := 0, ABS_INC := 0, ACC_SEL := 0, DEC_SEL := 0);
IF Axis4_DST.DONE THEN Run_Example := FALSE; END_IF;
(* Command to perform direct home of axes 1 and 4 *)
(* Rung L30 *)
_p1 := Home_Axes AND _0002_A1_RDY AND _0002_A4_RDY AND _0002_LINKUP_INFO;
Axis1_Home(REQ := _p1, BASE := 0, SLOT := 2, AXIS := 1);
Axis4_Home(REQ := _p1, BASE := 0, SLOT := 2, AXIS := 4);
IF Axis4_Home.DONE THEN Home_Axes := FALSE; END_IF;
(* Shows example of connecting to ECAT servo drives *)
(* Rung L43 *)
ECON_FB(REQ := Connect_Servos, BASE := 0, SLOT := 2);
IF ECON_FB.DONE THEN Connect_Servos := FALSE; END_IF;

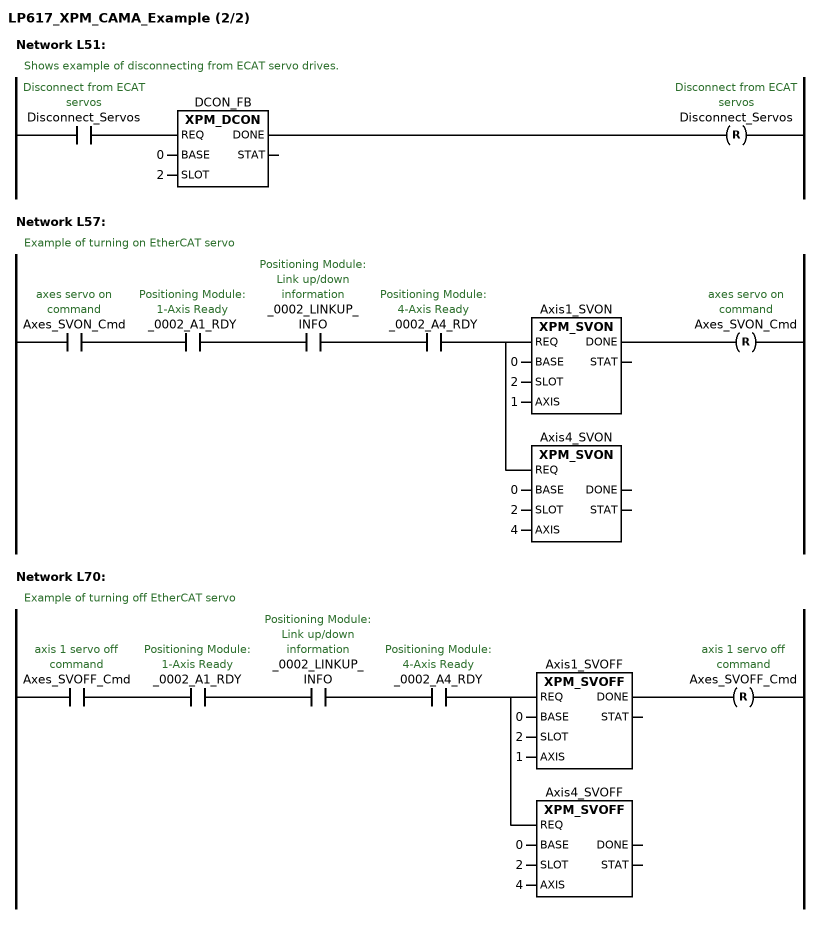
(* Shows example of disconnecting from ECAT servo drives. *)
(* Rung L51 *)
DCON_FB(REQ := Disconnect_Servos, BASE := 0, SLOT := 2);
IF DCON_FB.DONE THEN Disconnect_Servos := FALSE; END_IF;
(* Example of turning on EtherCAT servo *)
(* Rung L57 *)
_p2 := Axes_SVON_Cmd AND _0002_A1_RDY AND _0002_LINKUP_INFO AND _0002_A4_RDY;
Axis1_SVON(REQ := _p2, BASE := 0, SLOT := 2, AXIS := 1);
IF Axis1_SVON.DONE THEN Axes_SVON_Cmd := FALSE; END_IF;
Axis4_SVON(REQ := _p2, BASE := 0, SLOT := 2, AXIS := 4);
(* Example of turning off EtherCAT servo *)
(* Rung L70 *)
_p3 := Axes_SVOFF_Cmd AND _0002_A1_RDY AND _0002_LINKUP_INFO AND _0002_A4_RDY;
Axis1_SVOFF(REQ := _p3, BASE := 0, SLOT := 2, AXIS := 1);
IF Axis1_SVOFF.DONE THEN Axes_SVOFF_Cmd := FALSE; END_IF;
Axis4_SVOFF(REQ := _p3, BASE := 0, SLOT := 2, AXIS := 4);
END_PROGRAM

PROGRAM LP618_XPM_GEARIP_Example (* task: Scan Program *)
(* example program for XPM_GEARIP function block. *)
VAR
    Axes_SVOFF_Cmd : BOOL; (* axis 1 servo off command *)
    Axes_SVON_Cmd : BOOL; (* axes servo on command *)
    Axis1_GearIP : XPM_GEARIP; (* XPM_GEARIP fb for axis 1 *)
    Axis1_Home : XPM_FLT; (* direct home of axis 1 *)
    Axis1_SVOFF : XPM_SVOFF; (* function block for axis 1 servo off *)
    Axis1_SVON : XPM_SVON; (* SVON fb for axis 1 *)
    Axis1_Sync_CMD1 : BOOL; (* command to perform XPM_SSSD fb *)
    Axis4_DST : XPM_DST; (* direct start for axis 4 *)
    Axis4_Home : XPM_FLT; (* direct home axis 4 *)
    Axis4_SVOFF : XPM_SVOFF; (* servo off fb for axis 4 *)
    Axis4_SVON : XPM_SVON; (* servo on fb for axis 4 *)
    Connect_Servos : BOOL; (* command to connect to ECAT servos *)
    DCON_FB : XPM_DCON; (* EtherCAT disconnect FB *)
    Disconnect_Servos : BOOL; (* Disconnect from ECAT servos *)
    ECON_FB : XPM_ECON; (* EtherCAT connect FB *)
    Home_Axes : BOOL; (* home the axes *)
END_VAR
VAR_EXTERNAL
    _0002_A1_RDY : BOOL; (* AT %UX0.2.0 *) (* Positioning Module: 1-Axis Ready *)
    _0002_A4_RDY : BOOL; (* AT %UX0.2.3 *) (* Positioning Module: 4-Axis Ready *)
    _0002_LINKUP_INFO : BOOL; (* AT %UX0.2.14 *) (* Positioning Module: Link up/down information *)
END_VAR
VAR
    _p1 : BOOL;
    _p2 : BOOL;
    _p3 : BOOL;
END_VAR

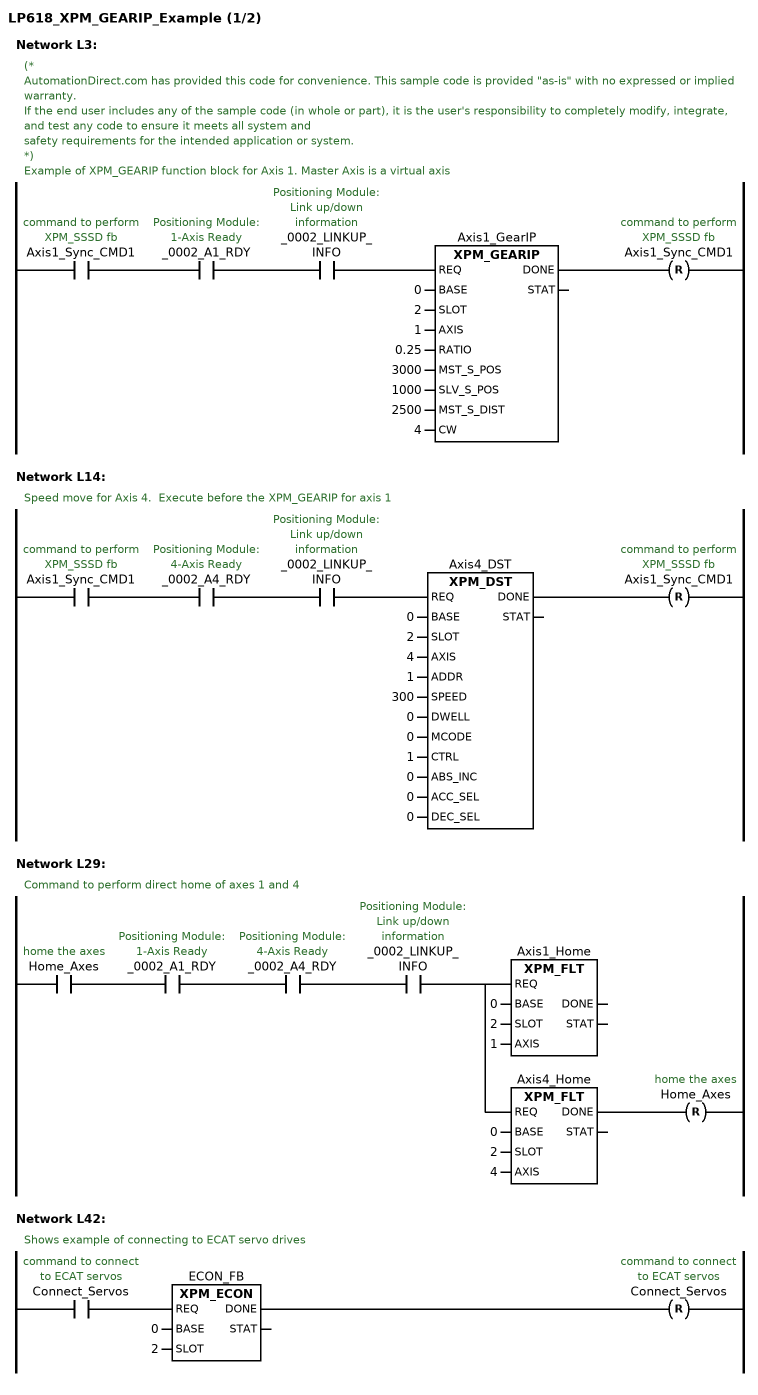
(* ( * / AutomationDirect.com has provided this code for convenience. This sample code is provided "as-is" with no expressed or implied warranty. / If the end user includes any of the sample code (in whole or part), it is the user's responsibility to completely modify, integrate, and test any code to ensure it meets all system and / safety requirements for the intended application or system. / * ) *)
(* Example of XPM_GEARIP function block for Axis 1. Master Axis is a virtual axis *)
(* Rung L3 *)
Axis1_GearIP(REQ := Axis1_Sync_CMD1 AND _0002_A1_RDY AND _0002_LINKUP_INFO, BASE := 0, SLOT := 2, AXIS := 1, RATIO := 0.25, MST_S_POS := 3000, SLV_S_POS := 1000, MST_S_DIST := 2500, CW := 4);
IF Axis1_GearIP.DONE THEN Axis1_Sync_CMD1 := FALSE; END_IF;
(* Speed move for Axis 4.  Execute before the XPM_GEARIP for axis 1 *)
(* Rung L14 *)
Axis4_DST(REQ := Axis1_Sync_CMD1 AND _0002_A4_RDY AND _0002_LINKUP_INFO, BASE := 0, SLOT := 2, AXIS := 4, ADDR := 1, SPEED := 300, DWELL := 0, MCODE := 0, CTRL := 1, ABS_INC := 0, ACC_SEL := 0, DEC_SEL := 0);
IF Axis4_DST.DONE THEN Axis1_Sync_CMD1 := FALSE; END_IF;
(* Command to perform direct home of axes 1 and 4 *)
(* Rung L29 *)
_p1 := Home_Axes AND _0002_A1_RDY AND _0002_A4_RDY AND _0002_LINKUP_INFO;
Axis1_Home(REQ := _p1, BASE := 0, SLOT := 2, AXIS := 1);
Axis4_Home(REQ := _p1, BASE := 0, SLOT := 2, AXIS := 4);
IF Axis4_Home.DONE THEN Home_Axes := FALSE; END_IF;
(* Shows example of connecting to ECAT servo drives *)
(* Rung L42 *)
ECON_FB(REQ := Connect_Servos, BASE := 0, SLOT := 2);
IF ECON_FB.DONE THEN Connect_Servos := FALSE; END_IF;

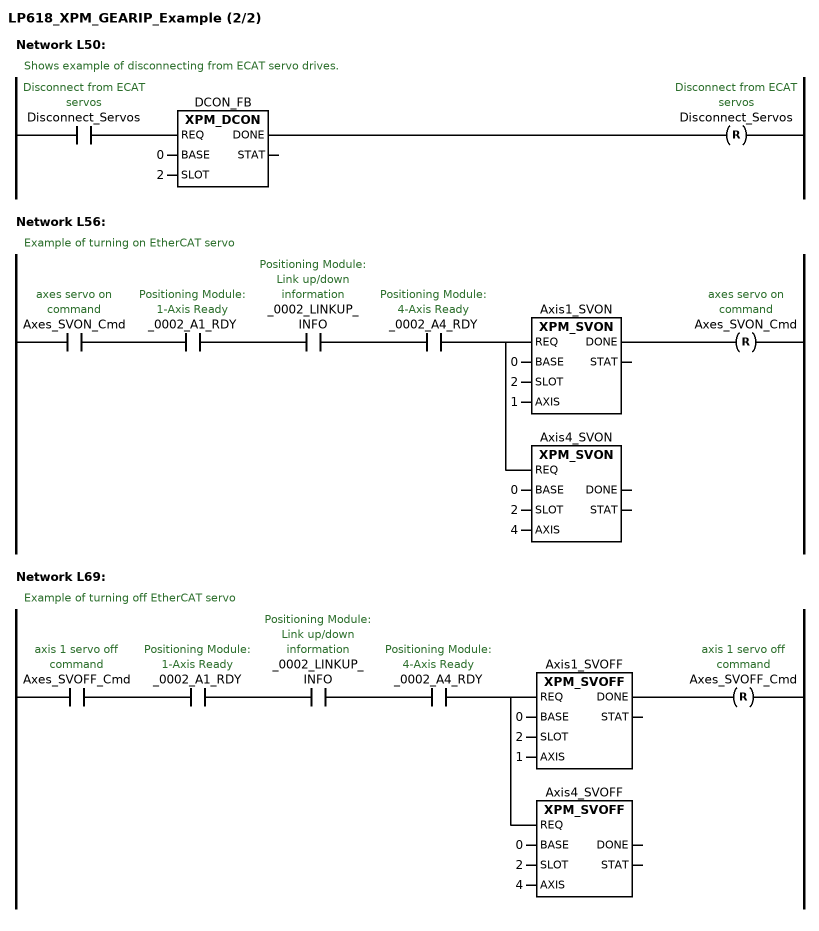
(* Shows example of disconnecting from ECAT servo drives. *)
(* Rung L50 *)
DCON_FB(REQ := Disconnect_Servos, BASE := 0, SLOT := 2);
IF DCON_FB.DONE THEN Disconnect_Servos := FALSE; END_IF;
(* Example of turning on EtherCAT servo *)
(* Rung L56 *)
_p2 := Axes_SVON_Cmd AND _0002_A1_RDY AND _0002_LINKUP_INFO AND _0002_A4_RDY;
Axis1_SVON(REQ := _p2, BASE := 0, SLOT := 2, AXIS := 1);
IF Axis1_SVON.DONE THEN Axes_SVON_Cmd := FALSE; END_IF;
Axis4_SVON(REQ := _p2, BASE := 0, SLOT := 2, AXIS := 4);
(* Example of turning off EtherCAT servo *)
(* Rung L69 *)
_p3 := Axes_SVOFF_Cmd AND _0002_A1_RDY AND _0002_LINKUP_INFO AND _0002_A4_RDY;
Axis1_SVOFF(REQ := _p3, BASE := 0, SLOT := 2, AXIS := 1);
IF Axis1_SVOFF.DONE THEN Axes_SVOFF_Cmd := FALSE; END_IF;
Axis4_SVOFF(REQ := _p3, BASE := 0, SLOT := 2, AXIS := 4);
END_PROGRAM

PROGRAM LP620_XPM_TRQSL_Example (* task: Scan Program *)
(* this is an example of XPM_TRQSL *)
VAR
    Axes_SVOFF_Cmd : BOOL; (* axis 1 servo off command *)
    Axes_SVON_Cmd : BOOL; (* axes servo on command *)
    Axis1_Home : XPM_FLT; (* direct home of axis 1 *)
    Axis1_SVOFF : XPM_SVOFF; (* function block for axis 1 servo off *)
    Axis1_SVON : XPM_SVON; (* SVON fb for axis 1 *)
    Axis1_Torque_Time : UINT; (* gradient time for axis 1 torque fb *)
    Axis1_Torque_Value : INT; (* torque value for axis 1 *)
    Axis1_Trq_Speed_Limit : UINT; (* speed limit for XPM_TRQSL fb *)
    Connect_Servos : BOOL; (* command to connect to ECAT servos *)
    DCON_FB : XPM_DCON; (* EtherCAT disconnect FB *)
    Disconnect_Servos : BOOL; (* Disconnect from ECAT servos *)
    ECON_FB : XPM_ECON; (* EtherCAT connect FB *)
    Execute_Torque_Control : BOOL; (* command to execute torque control *)
    Home_Axes : BOOL; (* home the axes *)
    TorqueCtrl_FB : XPM_TRQSL; (* torque control fb for axis 1 *)
END_VAR
VAR_EXTERNAL
    _0002_A1_RDY : BOOL; (* AT %UX0.2.0 *) (* Positioning Module: 1-Axis Ready *)
    _0002_A4_RDY : BOOL; (* AT %UX0.2.3 *) (* Positioning Module: 4-Axis Ready *)
    _0002_LINKUP_INFO : BOOL; (* AT %UX0.2.14 *) (* Positioning Module: Link up/down information *)
END_VAR

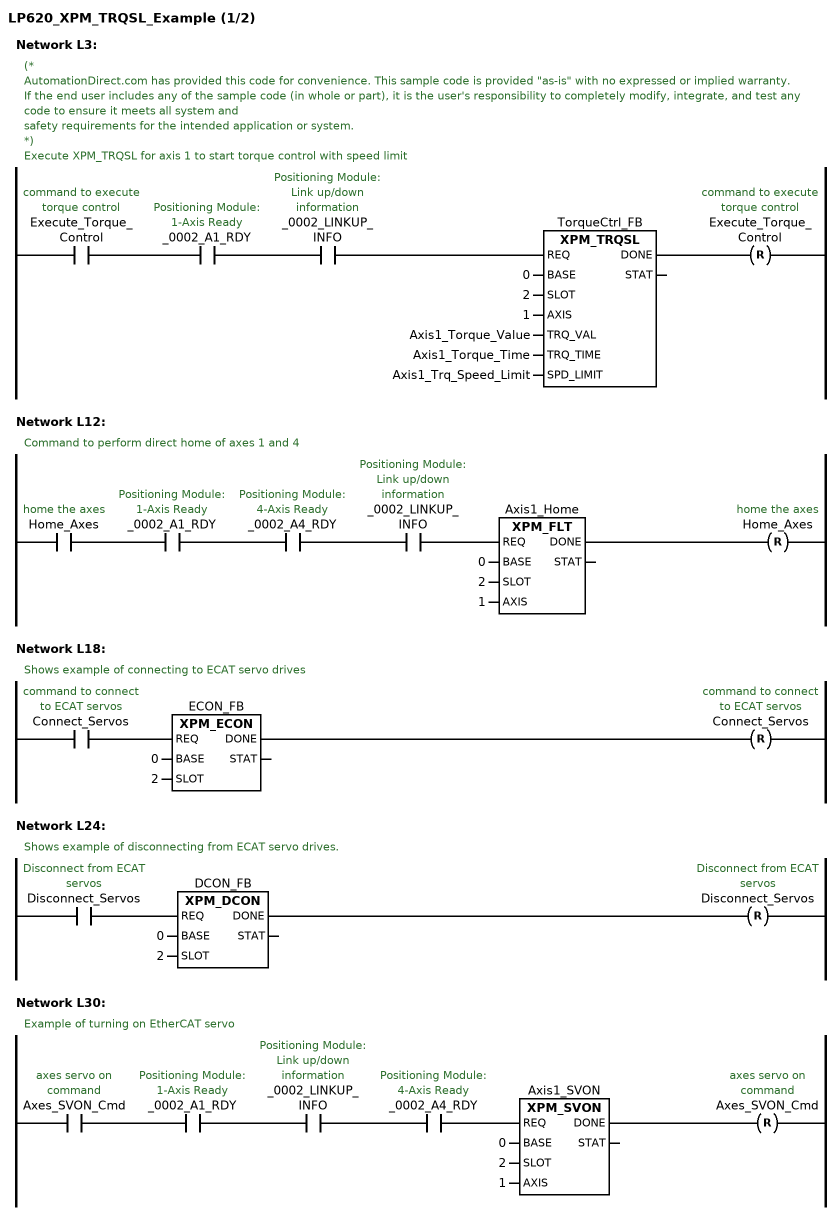
(* ( * / AutomationDirect.com has provided this code for convenience. This sample code is provided "as-is" with no expressed or implied warranty. / If the end user includes any of the sample code (in whole or part), it is the user's responsibility to completely modify, integrate, and test any code to ensure it meets all system and / safety requirements for the intended application or system. / * ) *)
(* Execute XPM_TRQSL for axis 1 to start torque control with speed limit *)
(* Rung L3 *)
TorqueCtrl_FB(REQ := Execute_Torque_Control AND _0002_A1_RDY AND _0002_LINKUP_INFO, BASE := 0, SLOT := 2, AXIS := 1, TRQ_VAL := Axis1_Torque_Value, TRQ_TIME := Axis1_Torque_Time, SPD_LIMIT := Axis1_Trq_Speed_Limit);
IF TorqueCtrl_FB.DONE THEN Execute_Torque_Control := FALSE; END_IF;
(* Command to perform direct home of axes 1 and 4 *)
(* Rung L12 *)
Axis1_Home(REQ := Home_Axes AND _0002_A1_RDY AND _0002_A4_RDY AND _0002_LINKUP_INFO, BASE := 0, SLOT := 2, AXIS := 1);
IF Axis1_Home.DONE THEN Home_Axes := FALSE; END_IF;
(* Shows example of connecting to ECAT servo drives *)
(* Rung L18 *)
ECON_FB(REQ := Connect_Servos, BASE := 0, SLOT := 2);
IF ECON_FB.DONE THEN Connect_Servos := FALSE; END_IF;
(* Shows example of disconnecting from ECAT servo drives. *)
(* Rung L24 *)
DCON_FB(REQ := Disconnect_Servos, BASE := 0, SLOT := 2);
IF DCON_FB.DONE THEN Disconnect_Servos := FALSE; END_IF;
(* Example of turning on EtherCAT servo *)
(* Rung L30 *)
Axis1_SVON(REQ := Axes_SVON_Cmd AND _0002_A1_RDY AND _0002_LINKUP_INFO AND _0002_A4_RDY, BASE := 0, SLOT := 2, AXIS := 1);
IF Axis1_SVON.DONE THEN Axes_SVON_Cmd := FALSE; END_IF;

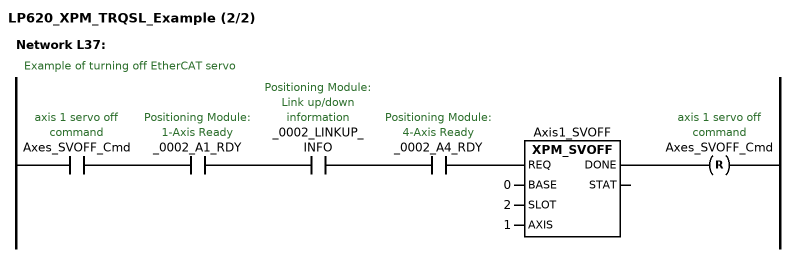
(* Example of turning off EtherCAT servo *)
(* Rung L37 *)
Axis1_SVOFF(REQ := Axes_SVOFF_Cmd AND _0002_A1_RDY AND _0002_LINKUP_INFO AND _0002_A4_RDY, BASE := 0, SLOT := 2, AXIS := 1);
IF Axis1_SVOFF.DONE THEN Axes_SVOFF_Cmd := FALSE; END_IF;
END_PROGRAM

PROGRAM LP621_XPM_TPROBE_ABORTT_Example (* task: Scan Program *)
(* example program for XPM_TPROBE and XPM_ABORTT  function blocks. *)
VAR
    Axes_SVOFF_Cmd : BOOL; (* axis 1 servo off command *)
    Axes_SVON_Cmd : BOOL; (* axes servo on command *)
    Axis1_Abortt_CMD : BOOL; (* execute Axis1 XPM_ABORTT *)
    Axis1_DST : XPM_DST; (* direct start for axis 4 *)
    Axis1_Home : XPM_FLT; (* direct home of axis 1 *)
    Axis1_LCLR_Cmd : BOOL; (* run latch clear position *)
    Axis1_LCNT : UINT; (* axis 1 l_cnt variable *)
    Axis1_LData : ARRAY[0..9] OF DINT; (* LDATA for axis 1 XPM_LRD fb *)
    Axis1_LRD_Cmd : BOOL; (* command to read latch position on axis 1 *)
    Axis1_Speed_CMD : BOOL; (* command to perform speed move of axis 1 *)
    Axis1_SVOFF : XPM_SVOFF; (* function block for axis 1 servo off *)
    Axis1_SVON : XPM_SVON; (* SVON fb for axis 1 *)
    Axis1_SVPWR : XPM_SVPWR; (* XPM_SVPWR fb *)
    Axis1_Tprobe2_CMD : BOOL; (* command for touch probe 2 *)
    Axis1_Tprobe_CMD : BOOL; (* execute XPM_TPROBE *)
    Axis1_XPM_ABORTT : XPM_ABORTT; (* XPM_ABORTT fb *)
    Axis1_XPM_LCLR : XPM_LCLR; (* axis 1 XPM_LCLR fb *)
    Axis1_XPM_LRD : XPM_LRD; (* axis 1 xpm_lrd fb *)
    Axis1_XPM_TPROBE1 : XPM_TPROBE; (* tprobe 1 fb *)
    Axis1_XPM_TPROBE2 : XPM_TPROBE; (* tprobe 2 fb *)
    Connect_Servos : BOOL; (* command to connect to ECAT servos *)
    DCON_FB : XPM_DCON; (* EtherCAT disconnect FB *)
    Disconnect_Servos : BOOL; (* Disconnect from ECAT servos *)
    ECON_FB : XPM_ECON; (* EtherCAT connect FB *)
    Execute_Parameter_Write : BOOL; (* command to write parameter data *)
    Home_Axes : BOOL; (* home the axes *)
    ParameterWrite_Data : DINT; (* data to write to a parameter *)
END_VAR
VAR_EXTERNAL
    _0002_A1_RDY : BOOL; (* AT %UX0.2.0 *) (* Positioning Module: 1-Axis Ready *)
    _0002_A4_RDY : BOOL; (* AT %UX0.2.3 *) (* Positioning Module: 4-Axis Ready *)
    _0002_LINKUP_INFO : BOOL; (* AT %UX0.2.14 *) (* Positioning Module: Link up/down information *)
END_VAR

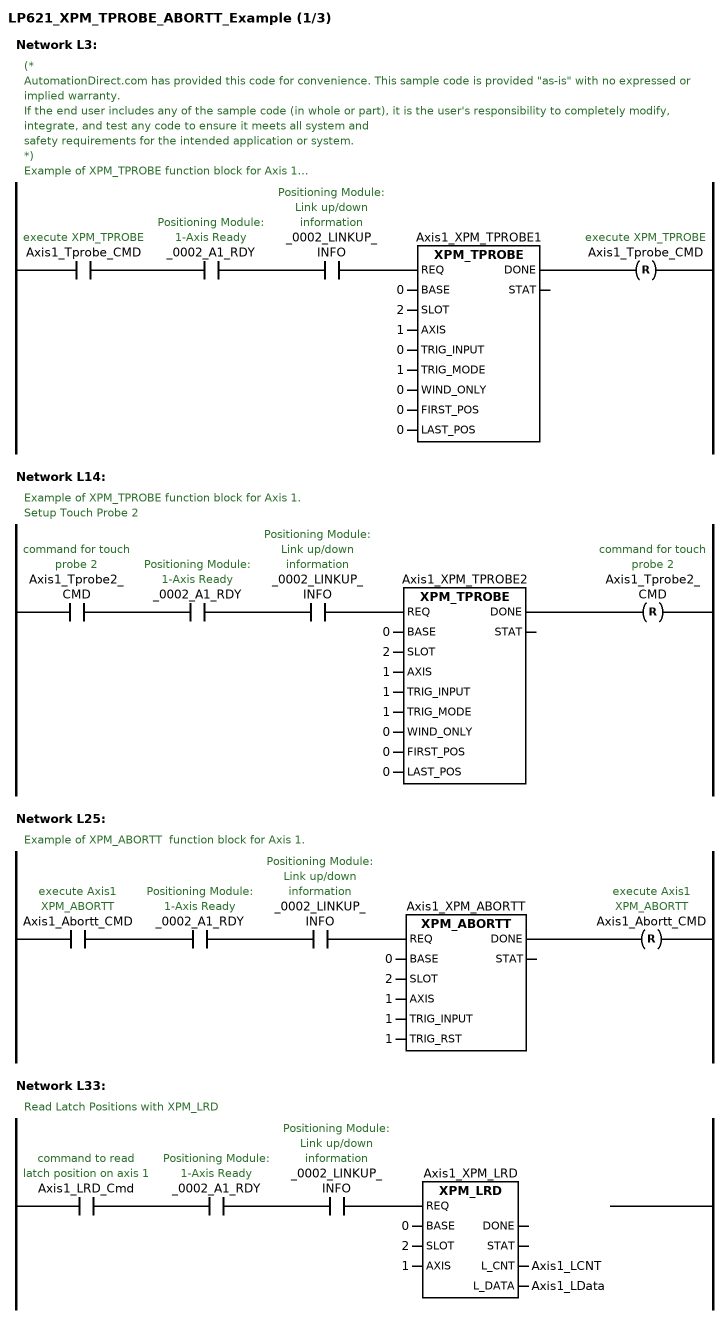
(* ( * / AutomationDirect.com has provided this code for convenience. This sample code is provided "as-is" with no expressed or implied warranty. / If the end user includes any of the sample code (in whole or part), it is the user's responsibility to completely modify, integrate, and test any code to ensure it meets all system and / safety requirements for the intended application or system. / * ) *)
(* Example of XPM_TPROBE function block for Axis 1. / Setup Touch Probe 1 *)
(* Rung L3 *)
Axis1_XPM_TPROBE1(REQ := Axis1_Tprobe_CMD AND _0002_A1_RDY AND _0002_LINKUP_INFO, BASE := 0, SLOT := 2, AXIS := 1, TRIG_INPUT := 0, TRIG_MODE := 1, WIND_ONLY := 0, FIRST_POS := 0, LAST_POS := 0);
IF Axis1_XPM_TPROBE1.DONE THEN Axis1_Tprobe_CMD := FALSE; END_IF;
(* Example of XPM_TPROBE function block for Axis 1. / Setup Touch Probe 2 *)
(* Rung L14 *)
Axis1_XPM_TPROBE2(REQ := Axis1_Tprobe2_CMD AND _0002_A1_RDY AND _0002_LINKUP_INFO, BASE := 0, SLOT := 2, AXIS := 1, TRIG_INPUT := 1, TRIG_MODE := 1, WIND_ONLY := 0, FIRST_POS := 0, LAST_POS := 0);
IF Axis1_XPM_TPROBE2.DONE THEN Axis1_Tprobe2_CMD := FALSE; END_IF;
(* Example of XPM_ABORTT  function block for Axis 1. *)
(* Rung L25 *)
Axis1_XPM_ABORTT(REQ := Axis1_Abortt_CMD AND _0002_A1_RDY AND _0002_LINKUP_INFO, BASE := 0, SLOT := 2, AXIS := 1, TRIG_INPUT := 1, TRIG_RST := 1);
IF Axis1_XPM_ABORTT.DONE THEN Axis1_Abortt_CMD := FALSE; END_IF;
(* Read Latch Positions with XPM_LRD *)
(* Rung L33 *)
Axis1_XPM_LRD(REQ := Axis1_LRD_Cmd AND _0002_A1_RDY AND _0002_LINKUP_INFO, BASE := 0, SLOT := 2, AXIS := 1, L_CNT => Axis1_LCNT, L_DATA => Axis1_LData);

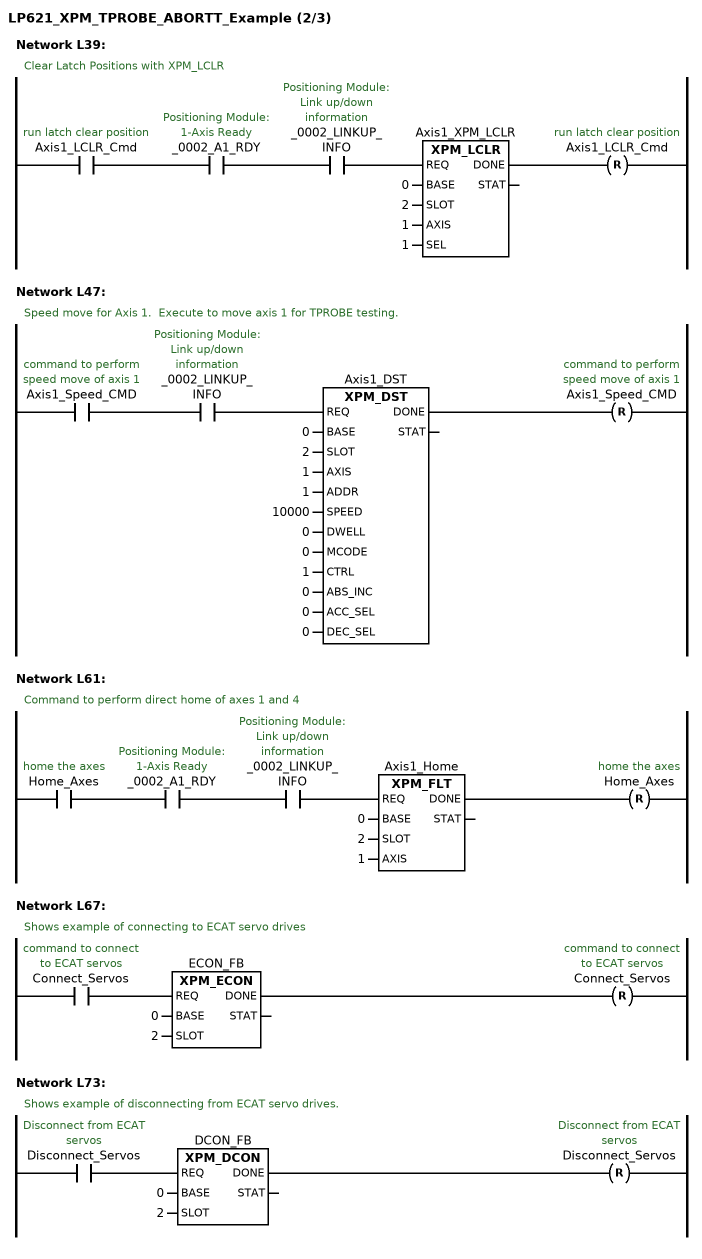
(* Clear Latch Positions with XPM_LCLR *)
(* Rung L39 *)
Axis1_XPM_LCLR(REQ := Axis1_LCLR_Cmd AND _0002_A1_RDY AND _0002_LINKUP_INFO, BASE := 0, SLOT := 2, AXIS := 1, SEL := 1);
IF Axis1_XPM_LCLR.DONE THEN Axis1_LCLR_Cmd := FALSE; END_IF;
(* Speed move for Axis 1.  Execute to move axis 1 for TPROBE testing. *)
(* Rung L47 *)
Axis1_DST(REQ := Axis1_Speed_CMD AND _0002_LINKUP_INFO, BASE := 0, SLOT := 2, AXIS := 1, ADDR := 1, SPEED := 10000, DWELL := 0, MCODE := 0, CTRL := 1, ABS_INC := 0, ACC_SEL := 0, DEC_SEL := 0);
IF Axis1_DST.DONE THEN Axis1_Speed_CMD := FALSE; END_IF;
(* Command to perform direct home of axes 1 and 4 *)
(* Rung L61 *)
Axis1_Home(REQ := Home_Axes AND _0002_A1_RDY AND _0002_LINKUP_INFO, BASE := 0, SLOT := 2, AXIS := 1);
IF Axis1_Home.DONE THEN Home_Axes := FALSE; END_IF;
(* Shows example of connecting to ECAT servo drives *)
(* Rung L67 *)
ECON_FB(REQ := Connect_Servos, BASE := 0, SLOT := 2);
IF ECON_FB.DONE THEN Connect_Servos := FALSE; END_IF;
(* Shows example of disconnecting from ECAT servo drives. *)
(* Rung L73 *)
DCON_FB(REQ := Disconnect_Servos, BASE := 0, SLOT := 2);
IF DCON_FB.DONE THEN Disconnect_Servos := FALSE; END_IF;

